# B&R Automation Studio project KeePak_Bliss_Reworked (part 2)

### Types.typ
```iecst
TYPE
	AdhesCtrlInterface_Commands_typ : 	STRUCT
		MelterOn : BOOL;
		MelterStandbyOff : BOOL;
		MelterStandbyOn : BOOL;
		PumpsOn : BOOL;
		PurgeChannel1 : {REDUND_UNREPLICABLE} BOOL;
		PurgeChannel2 : {REDUND_UNREPLICABLE} BOOL;
		PurgeChannel3 : {REDUND_UNREPLICABLE} BOOL;
		PurgeChannel4 : {REDUND_UNREPLICABLE} BOOL;
		WriteChannelTemp : BOOL;
		GlobalTempChanged : BOOL;
	END_STRUCT;
	AdhesCtrlInterface_Pars_typ : 	STRUCT
		SavedPatterns : ARRAY[0..3]OF AdhesivePatternCollections_typ;
		AdhesivePatterns : {REDUND_UNREPLICABLE} ARRAY[0..MAX_NUM_GLUE_CHANNELS_M1]OF AdhesivePattern_typ;
		AdhesiveHMIPatterns : {REDUND_UNREPLICABLE} ARRAY[0..MAX_NUM_GLUE_CHANNELS_M1]OF AdhesivePattern_typ;
		StitchPercentage : {REDUND_UNREPLICABLE} REAL;
		ChannelModulationCtrl : ARRAY[0..MAX_NUM_ONOFF_PATTERNS_M1]OF INT;
		BeadLengths : {REDUND_UNREPLICABLE} ARRAY[0..MAX_NUM_ONOFF_PATTERNS_M1]OF REAL := [4(10)];
		FeedbackIsHardwire : BOOL;
		FeedbackIsModbusTCP : BOOL;
		NordsonComms : NordsonData_typ;
		NordsonFeedbackSelection : NordsonFeedbackSelection_enum;
		NumAdhesiveChannels : {REDUND_UNREPLICABLE} USINT;
		PatternSelection : USINT;
	END_STRUCT;
	AdhesCtrlInterface_Status_typ : 	STRUCT
		AlarmActive : {REDUND_UNREPLICABLE} BOOL;
		ATS_AddOnOverLimit : BOOL;
		ATS_AddOnUnderLimit : BOOL;
		FeederFault : {REDUND_UNREPLICABLE} BOOL;
		GlueApplicationAllowed : {REDUND_UNREPLICABLE} BOOL;
		GlueCyclePos : {REDUND_UNREPLICABLE} REAL;
		LatchedEncoderPos : {REDUND_UNREPLICABLE} REAL;
		LowLevel : {REDUND_UNREPLICABLE} BOOL;
		NordsonInStandby : BOOL;
		ServiceNeeded : {REDUND_UNREPLICABLE} BOOL;
		UnitFault : {REDUND_UNREPLICABLE} BOOL;
		UnitReady : {REDUND_UNREPLICABLE} BOOL;
	END_STRUCT;
	AdhesiveChannelColormaps_typ : 	STRUCT
		Delay : {REDUND_UNREPLICABLE} ARRAY[0..MAX_NUM_ONOFF_PATTERNS_M1]OF USINT;
		Glue : {REDUND_UNREPLICABLE} ARRAY[0..MAX_NUM_ONOFF_PATTERNS_M1]OF USINT;
	END_STRUCT;
	AdhesiveChannelDatapoints_typ : 	STRUCT
		Delay : {REDUND_UNREPLICABLE} ARRAY[0..MAX_NUM_ONOFF_PATTERNS_M1]OF UINT;
		Glue : {REDUND_UNREPLICABLE} ARRAY[0..MAX_NUM_ONOFF_PATTERNS_M1]OF UINT;
		RowLabel : {REDUND_UNREPLICABLE} UINT;
	END_STRUCT;
	AdhesiveCtrlInterface_typ : 	STRUCT
		Commands : {REDUND_UNREPLICABLE} AdhesCtrlInterface_Commands_typ;
		Parameters : {REDUND_UNREPLICABLE} AdhesCtrlInterface_Pars_typ;
		Status : {REDUND_UNREPLICABLE} AdhesCtrlInterface_Status_typ;
	END_STRUCT;
	AdhesivePatternCollections_typ : 	STRUCT
		AdhesivePatterns : ARRAY[0..MAX_NUM_GLUE_CHANNELS_M1]OF AdhesivePattern_typ;
	END_STRUCT;
	AdhesivePattern_typ : 	STRUCT
		DelayDistance : {REDUND_UNREPLICABLE} ARRAY[0..MAX_NUM_ONOFF_PATTERNS_M1]OF REAL;
		GlueOnDistance : {REDUND_UNREPLICABLE} ARRAY[0..MAX_NUM_ONOFF_PATTERNS_M1]OF REAL;
	END_STRUCT;
	AlarmListAdapter_typ : 	STRUCT
		Acknowledged : {REDUND_UNREPLICABLE} ARRAY[0..49]OF STRING[10];
		Active : {REDUND_UNREPLICABLE} ARRAY[0..49]OF STRING[10];
		Code : {REDUND_UNREPLICABLE} ARRAY[0..49]OF STRING[10];
	END_STRUCT;
	AxisInitStates_enum :
		( (*Axis Control States*)
		AXIS_INIT_DONE := 500,
		AXIS_INIT_RETRIEVE_PARS := 10,
		AXIS_INIT_TRANSFER_PARS := 0,
		AXIS_INIT_WAIT_FOR_INIT := 20
		);
	AxisStates_enum :
		( (*Axis Control States*)
		AXIS_STATE_INIT := 0,
		AXIS_STATE_POWERON_PREP := 1,
		AXIS_STATE_POWERON := 2,
		AXIS_STATE_COUPLED := 70,
		AXIS_STATE_ERROR := 999,
		AXIS_STATE_HOME := 30,
		AXIS_STATE_IDLE := 80,
		AXIS_STATE_MOVE := 90,
		AXIS_STATE_MOVE_TO_MASTER := 50,
		AXIS_STATE_MOVE_VELOCITY := 91,
		AXIS_STATE_WAIT_FOR_MASTER_READY := 85,
		AXIS_STATE_W_COUPLE := 60,
		AXIS_STATE_W_HOME := 40,
		AXIS_STATE_POWERSAVER := 100,
		AXIS_STATE_POWERBACK := 101
		);
	Axis_enums :
		( (*Axis enumerations*)
		CCW := 4,
		CC_LEFT := 2,
		CC_RIGHT := 3,
		CSW_LEFT := 0,
		CSW_Left11 := 11,
		CSW_Left12 := 12,
		CSW_Left13 := 13,
		CSW_Left14 := 14,
		CSW_Left15 := 15,
		CSW_Left16 := 16,
		CSW_Left17 := 17,
		CSW_Left18 := 18,
		CSW_Left19 := 19,
		CSW_RIGHT := 1,
		FOLDING_ARM_DA_LEFT := 7,
		FOLDING_ARM_DA_RIGHT := 8,
		FOLDING_BAR := 5,
		FOLDING_TOOL_HA_LEFT := 9,
		FOLDING_TOOL_HA_RIGHT := 10,
		FTCL := 6
		);
	Axis_Interface_Comds_ToMapp_typ : 	STRUCT  (*Axis Commands to Mapp*)
		CoupleToMaster : BOOL;
		Home : BOOL;
		JogNeg : BOOL;
		JogPos : BOOL;
		LoadConfig : BOOL;
		MoveAbs : BOOL;
		MoveAdditive : BOOL;
		MoveVelocity : BOOL;
		Power : BOOL;
		SaveConfig : BOOL;
		Stop : BOOL;
		TorqueLimitingOn : BOOL;
		Update : BOOL;
	END_STRUCT;
	Axis_Interface_Commands_typ : 	STRUCT  (*Axis Commands*)
		Init : BOOL;
		MoveVelocityTrigStop : BOOL;
		RequestCoupleToMaster : BOOL;
		RequestHome : BOOL;
		RequestJogNeg : BOOL;
		RequestJogPos : BOOL;
		RequestMoveAbs : BOOL;
		RequestMoveAdditive : BOOL;
		RequestMoveVelocity : BOOL;
		Stop : USINT;
		ToMapp : Axis_Interface_Comds_ToMapp_typ;
		StartPowerSaver : BOOL;
		StopPowerSaver : BOOL;
	END_STRUCT;
	Axis_Interface_Parameters_typ : 	STRUCT  (*Axis Parameters*)
		AxisAndDrivePars : MpAxisBasicConfigType;
		CouplingMaster : UDINT;
		CouplingParameters : MpAxisCouplingParType;
		MovementParameters : MpAxisBasicParType;
		TriggerDistance : REAL; (*Distance that should be moved after an axis sees a tigger event when using MC_BR_MoveVelocityTriggStop*)
	END_STRUCT;
	Axis_Interface_Status_typ : 	STRUCT  (*Axis Statuses*)
		ActualTorque : LREAL;
		ActualPosition : LREAL;
		ActualSpeed : REAL;
		AxisInitialized : BOOL;
		AxisState : STRING[50];
		ConfigCommandDone : BOOL;
		DefaultRecipeLoaded : BOOL;
		Error : BOOL;
		Homed : BOOL;
		InMotion : BOOL;
		InPosition : BOOL;
		InSync : BOOL;
		MappCommandBusy : BOOL;
		MoveComplete : BOOL;
		PoweredOn : BOOL;
		ReadyToPowerOn : BOOL;
		TriggerMoveDone : BOOL;
		AxisBasicActive : BOOL;
		ClearOfRoller : BOOL;
		PositiveStatusID : USINT; (*The absolute value of the Info.Diag.StatusID.ID from the AxisBasic FUB*)
		StatusSeverity : UDINT;
		StatusCode : UINT;
		InternalID : DINT;
		InternalSeverity : UDINT;
		PositiveInternalFacility : UDINT; (*The absolute value of  Info.Diag.Internal.Facility from the AxisBasic FUB*)
		InternalCode : UINT;
		ExecutingCmd : UDINT;
		PowerSaverModeOn : BOOL;
	END_STRUCT;
	Axis_Interface_typ : 	STRUCT  (*servo Axis Interface*)
		Commands : Axis_Interface_Commands_typ;
		Parameters : Axis_Interface_Parameters_typ;
		Status : Axis_Interface_Status_typ;
	END_STRUCT;
	BitmapSelectDatapoints_typ : 	STRUCT
		AlarmActive : {REDUND_UNREPLICABLE} USINT;
		ResetPress : {REDUND_UNREPLICABLE} BOOL;
		RunPress : {REDUND_UNREPLICABLE} BOOL;
		StopPress : {REDUND_UNREPLICABLE} BOOL;
		VacuumPress : {REDUND_UNREPLICABLE} BOOL;
	END_STRUCT;
	Channel_typ : 	STRUCT
		ActualPressure : REAL;
		PressureSetpoint : REAL;
	END_STRUCT;
	ColorMapDatapoints_typ : 	STRUCT
		AdhesiveChannelsColormaps : {REDUND_UNREPLICABLE} ARRAY[0..MAX_NUM_GLUE_CHANNELS_M1]OF AdhesiveChannelColormaps_typ;
		AdhesiveSystemOK : {REDUND_UNREPLICABLE} USINT;
		AdhesiveUnitFault : {REDUND_UNREPLICABLE} USINT;
		AdhesiveUnitFeederFault : {REDUND_UNREPLICABLE} USINT;
		AdhesiveUnitLevelLow : {REDUND_UNREPLICABLE} USINT;
		AdhesiveUnitReady : {REDUND_UNREPLICABLE} USINT;
		AdhesiveUnitServiceNeeded : {REDUND_UNREPLICABLE} USINT;
		AdhesiveUseageLow : {REDUND_UNREPLICABLE} USINT;
		AirPressureOK : {REDUND_UNREPLICABLE} USINT;
		ATSAddOnOver : USINT;
		ATSAddOnUnder : USINT;
		AutoModeSelected : {REDUND_UNREPLICABLE} USINT;
		DownstreamSensorOK : {REDUND_UNREPLICABLE} USINT;
		DriveFaultOK : {REDUND_UNREPLICABLE} USINT;
		GlueSystemOK : {REDUND_UNREPLICABLE} USINT;
		JogModeSelected : {REDUND_UNREPLICABLE} USINT;
		NordsonEditTemps : USINT;
		RecipeLoaded : {REDUND_UNREPLICABLE} USINT;
		RecipeSystemBusy : {REDUND_UNREPLICABLE} USINT;
		SafetyOK : {REDUND_UNREPLICABLE} USINT;
		VacuumOK : {REDUND_UNREPLICABLE} USINT;
		VacuumPressureOK : {REDUND_UNREPLICABLE} USINT;
		VacuumPumpOn : {REDUND_UNREPLICABLE} USINT;
		Valve1OK : {REDUND_UNREPLICABLE} USINT;
		Valve2OK : {REDUND_UNREPLICABLE} USINT;
		Valve3OK : {REDUND_UNREPLICABLE} USINT;
		Valve4OK : USINT;
	END_STRUCT;
	DigitalInputs_typ : 	STRUCT
		AdhesiveLevelLow : {REDUND_UNREPLICABLE} BOOL;
		AdhesivePhotoEye : {REDUND_UNREPLICABLE} BOOL;
		AdhesivePhotoEye_2 : {REDUND_UNREPLICABLE} BOOL;
		AdhesiveUnitNotFaulted : {REDUND_UNREPLICABLE} BOOL;
		AdhesiveUnitReady : {REDUND_UNREPLICABLE} BOOL;
		AirPressureOK : {REDUND_UNREPLICABLE} BOOL;
		BodyDetect : BOOL;
		DownstreamSensor : {REDUND_UNREPLICABLE} BOOL;
		DownstreamSensorRaw : {REDUND_UNREPLICABLE} BOOL;
		LeftEndDetect : BOOL;
		LowAdhesiveUseage : {REDUND_UNREPLICABLE} BOOL;
		Pneumatics580StatusWord3 : {REDUND_UNREPLICABLE} UINT;
		PnuematicsHWStatusV0 : BOOL;
		PnuematicsHWStatusV2 : BOOL;
		PnuematicsHWStatusV4 : BOOL;
		PnuematicsHWStatusV6 : BOOL;
		RightEndDetect : BOOL;
		SafetyOK : {REDUND_UNREPLICABLE} BOOL;
		SSI_Parallel : {REDUND_UNREPLICABLE} SSI_Paraller_typ;
		VacHigh : BOOL;
		VacLow : BOOL;
		VacuumPressureOK : {REDUND_UNREPLICABLE} BOOL;
		VacuumTempOK : {REDUND_UNREPLICABLE} BOOL;
		X_PickRetracted : BOOL;
		X_PickExtended : BOOL;
		Y_PickRetract : BOOL;
		X_BlowOff : BOOL;
		BodyHopperLow : BOOL;
		LeftHopperLow : BOOL;
		RightHopperLow : BOOL;
		BodyHopperMotor_RUN : BOOL;
		LeftHopperMotor_RUN : BOOL;
		RightHopperMotor_RUN : BOOL;
		LubricationCounter : BOOL;
		BodyHopperMotor_OFF : BOOL;
		LeftHopperMotor_OFF : BOOL;
		RightHopperMotor_OFF : BOOL;
		DownstreamSensorON : BOOL;
		BodyPickHome : BOOL;
		BodyVacuumAchieved : BOOL;
		SidePickVacuumAchieved : BOOL;
		SideFoldSensor : BOOL;
		SideFoldVacuumAchieved : BOOL;
	END_STRUCT;
	DigitalOutputs_typ : 	STRUCT
		AirOn : {REDUND_UNREPLICABLE} BOOL;
		AmberLightStack : {REDUND_UNREPLICABLE} BOOL;
		BlowOffOn : BOOL;
		BottomFolder : {REDUND_UNREPLICABLE} BOOL;
		CompressionAirOn : BOOL;
		GlueChannel1 : {REDUND_UNREPLICABLE} BOOL;
		GlueChannel2 : {REDUND_UNREPLICABLE} BOOL;
		GlueChannel3 : {REDUND_UNREPLICABLE} BOOL;
		GlueChannel4 : {REDUND_UNREPLICABLE} BOOL;
		GreenLightStack : {REDUND_UNREPLICABLE} BOOL;
		HighCompression : BOOL;
		LowCompression : BOOL;
		PickAndPlace_X : BOOL;
		Pneumatics580ControlWord1 : {REDUND_UNREPLICABLE} UINT;
		PnuematicsValve0 : BOOL;
		PnuematicsValve2 : BOOL;
		PnuematicsValve4 : BOOL;
		PnuematicsValve6 : BOOL;
		PushOn : {REDUND_UNREPLICABLE} BOOL;
		RedLightStack : {REDUND_UNREPLICABLE} BOOL;
		ResetEuchner : BOOL;
		ResetSafety : {REDUND_UNREPLICABLE} BOOL;
		TopFolder : {REDUND_UNREPLICABLE} BOOL;
		VacuumOn : {REDUND_UNREPLICABLE} BOOL;
		ZeroEncoder : {REDUND_UNREPLICABLE} BOOL;
		SidePanelVacOn : BOOL;
		SidePanelVacBlowOff : BOOL;
		X_PickSolenoid : BOOL;
		Y_PickSolenoid : BOOL;
		OutConveyorOn_1 : BOOL;
		OutConveyorOn_2 : BOOL;
		OutConveyorOn_3 : BOOL;
		BodyVacuumOn : BOOL;
		BodyKicker : BOOL;
		SidePickCylinder : BOOL;
		LeftSideFoldCylinder : BOOL;
		RightSideFoldCylinder : BOOL;
		SidePanelHoldVacuum : BOOL;
		FoldingHoldVacuum : BOOL;
		CompressionCylinder : BOOL;
	END_STRUCT;
	Encoders_typ : {REDUND_UNREPLICABLE} 	STRUCT
		SickSSIPos : {REDUND_UNREPLICABLE} UDINT;
		SickSSIPosDegrees : {REDUND_UNREPLICABLE} REAL;
		FeedEncoderPos : {REDUND_UNREPLICABLE} UDINT;
		FeedEncoderPosDegrees : {REDUND_UNREPLICABLE} REAL;
		RamEncoderPos : {REDUND_UNREPLICABLE} UDINT;
		RamEncoderPosDegrees : {REDUND_UNREPLICABLE} REAL;
	END_STRUCT;
	FolderTypeSelection_enum :
		(
		FOLDER_LINMOT := 1,
		FOLDER_PNEUMATIC := 0
		);
	FoldpushCtrlInterface_Pars_typ : 	STRUCT
		BottomFolderOffPos : REAL;
		BottomFolderOnPos : REAL;
		FolderTypeSelection : FolderTypeSelection_enum;
		HighCompressionOffPos : REAL;
		HighCompressionOnPos : REAL;
		LinMotBotFolder : LinAxis_typ;
		LinMotTopFolder : LinAxis_typ;
		LowCompressionOffPos : REAL;
		LowCompressionOnPos : REAL;
		NumaticsTypeSelection : NumaticsTypeSelection_enum;
		PushOff : {REDUND_UNREPLICABLE} REAL;
		PushOn : {REDUND_UNREPLICABLE} REAL;
		TopFolderOffPos : REAL;
		TopFolderOnPos : REAL;
	END_STRUCT;
	FoldpushCtrlInterface_Status_typ : 	STRUCT
		BottomFoldValveStatus : {REDUND_UNREPLICABLE} BOOL;
		CompOnValveStatus : BOOL;
		CompressionAllowed : BOOL;
		FoldersActuationAllowed : {REDUND_UNREPLICABLE} BOOL;
		HardwireConfig : BOOL;
		LinMotConfig : BOOL;
		PneumaticConfig : BOOL;
		PowelinkConfig : BOOL;
		PushValveStatus : {REDUND_UNREPLICABLE} BOOL;
		TopFoldValveStatus : {REDUND_UNREPLICABLE} BOOL;
	END_STRUCT;
	FoldPushCtrlInterface_typ : 	STRUCT
		Commands : {REDUND_UNREPLICABLE} FoldPushCtrlInt_Commands_typ;
		Parameters : {REDUND_UNREPLICABLE} FoldpushCtrlInterface_Pars_typ;
		Status : {REDUND_UNREPLICABLE} FoldpushCtrlInterface_Status_typ;
	END_STRUCT;
	FoldPushCtrlInt_Commands_typ : 	STRUCT
		placehold : {REDUND_UNREPLICABLE} BOOL;
	END_STRUCT;
	HMIControl_Commands_typ : 	STRUCT
		CancelBoxChange : BOOL;
		ConfirmBoxChange : BOOL;
		CycleBodyHopper : BOOL;
		CycleLeftHopper : BOOL;
		CycleRightHopper : BOOL;
		CycleServoRam : BOOL;
		CycleServoPnP : BOOL;
		HomeServoFeed : BOOL;
		HomeBodyHopper : BOOL;
		HomeLeftHopper : BOOL;
		HomeRightHopper : BOOL;
		HomeServoRam : BOOL;
		HomeServoPnP : BOOL;
		JogForward : BOOL;
		JogReverse : BOOL;
		JogServoFeedNeg : BOOL;
		JogServoFeedPos : BOOL;
		JogBodyHopperNeg : BOOL;
		JogBodyHopperPos : BOOL;
		JogLeftHopperNeg : BOOL;
		JogLeftHopperPos : BOOL;
		JogRightHopperNeg : BOOL;
		JogRightHopperPos : BOOL;
		JogServoRamNeg : BOOL;
		JogServoRamPos : BOOL;
		JogServoPnPNeg : BOOL;
		JogServoPnPPos : BOOL;
		LoadRecipe : BOOL;
		LoadRecipeType1 : BOOL;
		LoadRecipeType2 : BOOL;
		RequestBoxType1 : BOOL;
		RequestBoxType2 : BOOL;
		RequestReset : BOOL;
		RequestStop : BOOL;
		RequestVacuumOn : BOOL;
		RequestVFDRun : BOOL;
		SaveRecipe : BOOL;
		SelectAutoMode : BOOL;
		SelectJogMode : BOOL;
		StartServoFeed : BOOL;
		StartBodyHopper : BOOL;
		StartLeftHopper : BOOL;
		StartRightHopper : BOOL;
		ZeroEncoder : BOOL;
		EnableShowMode : BOOL;
	END_STRUCT;
	HMIControl_Parameters_typ : 	STRUCT
		ServoFeedAccel : REAL;
		ServoFeedJogVelocity : REAL;
		ServoFeedTorqueLimit : REAL;
		ServoFeedVelocity : REAL;
		BodyHopperAccel : REAL;
		BodyHopperEndDwellTime : UDINT;
		BodyHopperEndPosition : REAL;
		BodyHopperJogVelocity : REAL;
		BodyHopperStartDwellTime : UDINT;
		BodyHopperStartPosition : REAL;
		BodyHopperTorqueLimit : REAL;
		BodyHopperVelocity : REAL;
		BodyKickerTime : UDINT;
		BodyKickerRetractTime : UDINT;
		LeftHopperAccel : REAL;
		LeftHopperEndDwellTime : UDINT;
		LeftHopperEndPosition : REAL;
		LeftHopperJogVelocity : REAL;
		LeftHopperStartDwellTime : UDINT;
		LeftHopperStartPosition : REAL;
		LeftHopperTorqueLimit : REAL;
		LeftHopperVelocity : REAL;
		RightHopperAccel : REAL;
		RightHopperEndDwellTime : UDINT;
		RightHopperEndPosition : REAL;
		RightHopperJogVelocity : REAL;
		RightHopperStartDwellTime : UDINT;
		RightHopperStartPosition : REAL;
		RightHopperTorqueLimit : REAL;
		RightHopperVelocity : REAL;
		ServoRamAccel : REAL;
		ServoRamEndDwellTime : UDINT;
		ServoRamSidePickTime : UDINT;
		ServoRamSidePickRetractTime : UDINT;
		ServoRamSideFoldTime : UDINT;
		ServoRamSideFoldRetractTime : UDINT;
		ServoRamEndPosition : REAL;
		ServoRamFoldStartPos : REAL;
		ServoRamFoldEndPos : REAL;
		ServoRamJogVelocity : REAL;
		ServoRamStartDwellTime : UDINT;
		ServoRamStartPosition : REAL;
		ServoRamTorqueLimit : REAL;
		ServoRamNegativeVelocity : REAL;
		ServoRamSideFormingVelocity : REAL;
		ServoRamBoxFormingVelocity : REAL;
		ServoRamClearPosition : REAL;
		ServoRamMiddlePosition : REAL;
		ServoPnPAccel : REAL;
		ServoPnPEndDwellTime : UDINT;
		ServoPnPEndPosition : REAL;
		ServoPnPVacuumOffPosition : REAL;
		ServoPnPJogVelocity : REAL;
		ServoPnPStartDwellTime : UDINT;
		ServoPnPStartPosition : REAL;
		ServoPnPTorqueLimit : REAL;
		ServoPnPNegativeVelocity : REAL;
		ServoPnPPositiveVelocity : REAL;
		PickAndPlaceDwell : UDINT;
		BodyHopperDwellTime : UDINT;
		LeftHopperDwellTime : UDINT;
		RightHopperDwellTime : UDINT;
		BodyHopperTimeoutTime : UDINT;
		LeftHopperTimeoutTime : UDINT;
		RightHopperTimeoutTime : UDINT;
		ServoRamTimeoutTime : UDINT;
		ServoRamPowerSaverTime : UDINT;
		AtTorqueTime : UDINT;
		PickDwellTime : UDINT;
		TopFeedJamTime : UDINT;
		VacuumOffTime : UDINT;
		DownPulseTime : UDINT;
		Y_DelayTime : UDINT;
		BlowOffTime : UDINT;
		SetCycleCount : UDINT;
		LubeCycleCount : UDINT;
		LowFeedJamTime : UDINT;
		LowHopperTime : UDINT;
		LowBodyHopperTime : UDINT;
		LowLeftHopperTime : UDINT;
		LowRightHopperTime : UDINT;
		RamDelay : UDINT;
	END_STRUCT;
	HMIControl_typ : 	STRUCT
		BitmapSelectDatapoints : {REDUND_UNREPLICABLE} BitmapSelectDatapoints_typ;
		ColorMapDatapoints : {REDUND_UNREPLICABLE} ColorMapDatapoints_typ;
		Commands : {REDUND_UNREPLICABLE} HMIControl_Commands_typ;
		Parameters : HMIControl_Parameters_typ;
		StatusDatapoints : {REDUND_UNREPLICABLE} StatusDatapoints_typ;
	END_STRUCT;
	Home_Parameters_typ : 	STRUCT  (*Axis Homing Parameters*)
		ServoFeed : MpAxisHomingType;
		BodyHopper : MpAxisHomingType;
		LeftHopper : MpAxisHomingType;
		RightHopper : MpAxisHomingType;
		ServoRam : MpAxisHomingType;
		ServoPnP : MpAxisHomingType;
	END_STRUCT;
	IO_typ : 	STRUCT
		DIs : {REDUND_UNREPLICABLE} DigitalInputs_typ;
		DOs : {REDUND_UNREPLICABLE} DigitalOutputs_typ;
		Encoders : {REDUND_UNREPLICABLE} Encoders_typ;
		ModuleOKs : {REDUND_UNREPLICABLE} ARRAY[0..99]OF BOOL;
		SafetyStatus : SafetyStatus_typ;
	END_STRUCT;
	LightStack_typ :
		(
		LIGHTSTACK_PATLITE := 1,
		LIGHTSTACK_TRI := 0
		);
	LinAxisCommand_typ : 	STRUCT  (*Axis command type*)
		ErrorReset : BOOL; (*Reset error command*)
		Home : BOOL; (*Home command*)
		HomeRequest : BOOL; (*Request for home from HMI*)
		JogNegative : BOOL; (*Jog neg command*)
		JogNegativeRequest : BOOL; (*Request for jog negative*)
		JogPositive : BOOL; (*Jog pos command*)
		JogPositiveRequest : BOOL; (*Request for jog positive*)
		MoveAbsolute : BOOL; (*Move absolute command*)
		MoveAbsoluteRequest : BOOL; (*Request for move absolute*)
		MoveAdditive : BOOL; (*Move additive command*)
		Power : BOOL; (*Power command*)
		SaveConfig : BOOL;
		Stop : BOOL; (*Stop command*)
	END_STRUCT;
	LinAxisParameter_typ : 	STRUCT  (*Axis parameter type*)
		ExtendAccel : REAL;
		ExtendDecel : REAL;
		ExtendPos : LREAL;
		ExtendSpeed : REAL;
		MpBasicConfig : MpAxisBasicConfigType; (*Axis configuration parameters for change at runtime*)
		MpBasicParameters : MpAxisBasicParType; (*Mp params*)
		RetractAccel : REAL;
		RetractDecel : REAL;
		RetractPos : LREAL;
		RetractSpeed : REAL;
	END_STRUCT;
	LinAxisStatus_typ : 	STRUCT  (*Axis status type*)
		EndlessPosValid : BOOL; (*Endless position is valid*)
		Error : BOOL; (*Error active on axis*)
		ErrorId : DINT; (*Error id*)
		HomeCheck : BOOL;
		Info : MpAxisBasicInfoType;
		InPosition : BOOL; (*Axis in position*)
		IsHomed : BOOL; (*Axis is homed*)
		MoveActive : BOOL; (*Move is active on the axis*)
		Position : LREAL; (*Current position of axis*)
		PowerOn : BOOL; (*Axis is on*)
		Ready : BOOL; (*Axis is in standstill and homed*)
		Stopped : BOOL; (*Axis is stopped*)
		Velocity : REAL; (*Current velocity of axis*)
	END_STRUCT;
	LinAxis_typ : 	STRUCT  (*Axis type*)
		Command : LinAxisCommand_typ; (*Command*)
		Parameter : LinAxisParameter_typ; (*Parameter*)
		Status : LinAxisStatus_typ; (*Status*)
	END_STRUCT;
	LinMotState_enum :
		(
		STATE_ERROR,
		STATE_HOME_CHECK,
		STATE_HOME_RESTORE,
		STATE_HOME_STANDBY,
		STATE_HOME_TORQUE,
		STATE_INIT,
		STATE_IS_HOMED,
		STATE_JOG_NEG,
		STATE_JOG_POS,
		STATE_MOVE,
		STATE_READY
		);
	ModeCtrlInterface_Commands_typ : {REDUND_UNREPLICABLE} 	STRUCT
		ForceSafetyReset : {REDUND_UNREPLICABLE} BOOL;
		Reset : {REDUND_UNREPLICABLE} BOOL;
		Run : {REDUND_UNREPLICABLE} BOOL;
		SetAutoMode : {REDUND_UNREPLICABLE} BOOL;
		SetJogMode : {REDUND_UNREPLICABLE} BOOL;
		Stop : {REDUND_UNREPLICABLE} BOOL;
		SetShowMode : {REDUND_UNREPLICABLE} BOOL;
	END_STRUCT;
	ModeCtrlInterface_Parameters_typ : 	STRUCT
		BottomSensor : BOOL;
		DownstreamClear : UDINT := 1000;
		DownstreamIgnored : BOOL;
		DownstreamTimeout : UDINT := 1000;
		DwellTime : {REDUND_UNREPLICABLE} UDINT;
		InPositionTolerance : REAL := 10.0;
		LightStackSelection : LightStack_typ;
		MachineType : USINT;
		MaxPPM : UINT;
		MinPPM : UINT;
		PiecesPerMinute : {REDUND_UNREPLICABLE} UINT;
		SideSensors : BOOL;
		StopPosition : {REDUND_UNREPLICABLE} REAL;
		VaccumStopTime : UDINT := 200;
		SidePickTime : UDINT;
	END_STRUCT;
	ModeCtrlInterface_Status_typ : 	STRUCT
		AtStopPosition : {REDUND_UNREPLICABLE} BOOL;
		BlissPanelAlarmActive : BOOL;
		Dwelling : {REDUND_UNREPLICABLE} BOOL;
		DwellModeEnabled : {REDUND_UNREPLICABLE} BOOL;
		InAutoMode : {REDUND_UNREPLICABLE} BOOL;
		InBlissPanelWindow : BOOL;
		Jogging : {REDUND_UNREPLICABLE} BOOL;
		MachineIsBliss : BOOL;
		Running : {REDUND_UNREPLICABLE} BOOL;
		WaitingOnDownstream : BOOL;
	END_STRUCT;
	ModeCtrlInterface_typ : 	STRUCT
		Commands : {REDUND_UNREPLICABLE} ModeCtrlInterface_Commands_typ;
		Parameters : {REDUND_UNREPLICABLE} ModeCtrlInterface_Parameters_typ;
		Status : ModeCtrlInterface_Status_typ;
	END_STRUCT;
	NordsonData_typ : 	STRUCT
		AdhesiveUsePerHour : UDINT;
		Alert : BOOL;
		ByPassFeedback : BOOL;
		ChannelActTemp : ARRAY[0..NUM_NORDSON_TEMP_ZONES_M1]OF UINT;
		ChannelDataCmpResult : DINT;
		ChannelDataSize : UDINT;
		ChannelSetTempActual : ARRAY[0..NUM_NORDSON_TEMP_ZONES_M1]OF UINT;
		ChannelSetTempRequested : ARRAY[0..NUM_NORDSON_TEMP_ZONES_M1]OF UINT;
		CommFault : BOOL;
		CommFaultInDataValue : BOOL;
		ConsecutiveErrorCount : USINT;
		FeedbackTime : TIME := T#1s;
		HeatUpPhaseActive : BOOL;
		HoseSetTemp : UINT;
		MelterIsOn : BOOL;
		MelterStatus : UINT;
		PumpStartUpProtectionOn : BOOL;
		ShutDown : BOOL;
		StandbyTimeoutTime : TIME := T#2h;
		TempUnit : USINT;
		UnitFaulted : BOOL;
		UnitReady : BOOL;
		GlobalSetTemp : UINT;
	END_STRUCT;
	NordsonFeedbackSelection_enum :
		(
		NORDSON_HARDWIRE := 0,
		NORDSON_MODBUSTCP := 1
		);
	NordsonRxPacket_typ : 	STRUCT
		Byte0_1_Status : UINT;
		Byte2_Ack_Data_Index : USINT;
		Byte3_Ack_Channel_Num : USINT;
		Byte4_5_Read_Data_0 : UINT;
		Byte6_7_Read_Data_1 : UINT;
		Byte8_9_Read_Data_2 : UINT;
		Byte10_11_Read_Data_3 : UINT;
		Byte12_13_Read_Data_4 : UINT;
		Byte14_15_Read_Data_5 : UINT;
	END_STRUCT;
	NordsonTxPacket_typ : 	STRUCT
		Byte0_MelterControl : USINT;
		Byte1_Command : USINT;
		Byte2_Data_Index : USINT;
		Byte3_Channel_Num : USINT;
		Byte4_5_WriteData : UINT;
		Byte6_7_Mot1Spd : UINT;
		Byte8_9_Mot2Spd : UINT;
		Byte10_11_Mot3Spd : UINT;
		Byte12_13_Mot4Spd : UINT;
		Byte14_15_NotUsed : UINT;
	END_STRUCT;
	NumaticsTypeSelection_enum :
		(
		NUMATICS_HARDWIRE,
		NUMATICS_POWERLINK
		);
	RamControlInterface_typ : 	STRUCT
		Commands : {REDUND_UNREPLICABLE} RamCtrlInterface_Commands_typ;
		Parameters : {REDUND_UNREPLICABLE} RamCtrlInterface_Parameters_typ;
		Status : {REDUND_UNREPLICABLE} RamCtrlInterface_Status_typ;
	END_STRUCT;
	RamCtrlInterface_Commands_typ : 	STRUCT
		Home : {REDUND_UNREPLICABLE} BOOL;
		JogNegative : {REDUND_UNREPLICABLE} BOOL;
		JogPositive : {REDUND_UNREPLICABLE} BOOL;
		MoveAbsolute : {REDUND_UNREPLICABLE} BOOL;
		MoveAdditive : {REDUND_UNREPLICABLE} BOOL;
		MoveVelocity : {REDUND_UNREPLICABLE} BOOL;
		PowerOn : {REDUND_UNREPLICABLE} BOOL;
		VFDAlarmReset : {REDUND_UNREPLICABLE} BOOL;
	END_STRUCT;
	RamCtrlInterface_Parameters_typ : 	STRUCT
		Acceleration : {REDUND_UNREPLICABLE} REAL;
		CurrentLimit : {REDUND_UNREPLICABLE} REAL;
		GearRatio : REAL := 54;
		JogSpeed : {REDUND_UNREPLICABLE} REAL;
		Position : {REDUND_UNREPLICABLE} REAL;
	END_STRUCT;
	RamCtrlInterface_Status_typ : 	STRUCT
		ActualPosition : {REDUND_UNREPLICABLE} LREAL;
		ActualSpeed : {REDUND_UNREPLICABLE} LREAL;
		AlarmActive : {REDUND_UNREPLICABLE} BOOL;
		DriveSpeed : {REDUND_UNREPLICABLE} INT;
		Home : {REDUND_UNREPLICABLE} BOOL;
		InPosition : {REDUND_UNREPLICABLE} BOOL;
		MotorCurrent : {REDUND_UNREPLICABLE} UINT;
		MoveActive : {REDUND_UNREPLICABLE} BOOL;
		Position : {REDUND_UNREPLICABLE} REAL;
		PoweredOn : {REDUND_UNREPLICABLE} BOOL;
		Running : {REDUND_UNREPLICABLE} BOOL;
		Stopped : BOOL;
		STOStatus : UINT;
		VFDAlarmDetected : {REDUND_UNREPLICABLE} BOOL;
		VFDAlarmNumber : {REDUND_UNREPLICABLE} INT;
		VFDAlarmText : {REDUND_UNREPLICABLE} STRING[80];
	END_STRUCT;
	RecipeCtrlInterface_Commands_typ : 	STRUCT
		ChangeRecipe : BOOL;
		LoadRecipe : {REDUND_UNREPLICABLE} BOOL;
		SaveRecipe : {REDUND_UNREPLICABLE} BOOL;
	END_STRUCT;
	RecipeCtrlInterface_Pars_typ : 	STRUCT
		RecipeIndex : USINT;
		RecipeName : {REDUND_UNREPLICABLE} STRING[100];
	END_STRUCT;
	RecipeCtrlInterface_Status_typ : 	STRUCT
		Busy : {REDUND_UNREPLICABLE} BOOL;
		LoadedRecipeIndex : USINT;
		LoadedRecipeName : {REDUND_UNREPLICABLE} STRING[255];
		RecipeHasBeenLoaded : BOOL;
	END_STRUCT;
	RecipeCtrlInterface_typ : 	STRUCT
		Commands : {REDUND_UNREPLICABLE} RecipeCtrlInterface_Commands_typ;
		Parameters : {REDUND_UNREPLICABLE} RecipeCtrlInterface_Pars_typ;
		Status : {REDUND_UNREPLICABLE} RecipeCtrlInterface_Status_typ;
	END_STRUCT;
	Register_typ : 	STRUCT
		ChannelActualPressureWord : UDINT;
		ChannelSetPressureWord : UDINT;
		TankActualLevelWord : UINT;
	END_STRUCT;
	SafetyStatus_typ : 	STRUCT
		BackEstopOK : BOOL;
		CabinetEStopStatus : UINT;
		FrontEStopOK : BOOL;
		GuardDoorsOK : BOOL;
		SafetyProgramRunning : BOOL;
	END_STRUCT;
	SSI_Paraller_typ : {REDUND_UNREPLICABLE} 	STRUCT
		Bits : {REDUND_UNREPLICABLE} ARRAY[0..15]OF BOOL;
		FeedBits : {REDUND_UNREPLICABLE} ARRAY[0..15]OF BOOL;
		RamBits : {REDUND_UNREPLICABLE} ARRAY[0..15]OF BOOL;
	END_STRUCT;
	StatusDatapoints_typ : 	STRUCT
		AdhesiveChannelSDPs : {REDUND_UNREPLICABLE} ARRAY[0..MAX_NUM_GLUE_CHANNELS_M1]OF AdhesiveChannelDatapoints_typ;
		AdhesivePatternDialogSDP : UINT := 1;
		AdhesivePatternConfirmDialogSDP : UINT := 1;
		AdhesivePatternConfirmedSDP : UINT;
		AdhesiveUnitFaultSDP : {REDUND_UNREPLICABLE} UINT;
		AdhesiveUnitLevelLowSDP : {REDUND_UNREPLICABLE} UINT;
		AdhesiveUnitNotReadySDP : {REDUND_UNREPLICABLE} UINT;
		AdhesiveUseageLowSDP : {REDUND_UNREPLICABLE} UINT;
		AutoModeSDP : {REDUND_UNREPLICABLE} UINT;
		BlissSDP : UINT;
		HardwireValveSDP : USINT;
		JogStatusDatapoint : {REDUND_UNREPLICABLE} UINT;
		LinMotBotHomeSDP : UINT;
		LinMotSDP : UINT;
		LinMotTopHomeSDP : UINT;
		LinMotTuningSDP : UINT;
		MaintenanceSDP : {REDUND_UNREPLICABLE} UINT;
		MotorVacuumSDP : UINT;
		NordsonModbusSDP : UINT;
		NordsonStandbyOffSDP : UINT;
		PnuematicFolderSDP : UINT;
		RecipeDialogSDP : UINT;
		RecipeIndexSDP : UINT;
		RecipeReq1SDP : UINT;
		RecipeReq2SDP : UINT;
		RestartInhibitSDP : UINT;
		SafetyStartingSDP : UINT;
		ServoLayerSDP : {REDUND_UNREPLICABLE} UINT;
		ServoRamHomeSDP : UINT;
		SmartVacuumLayerSDP : {REDUND_UNREPLICABLE} UINT;
		TraySDP : UINT;
		VacuumPressureFaultSDP : {REDUND_UNREPLICABLE} UINT;
		VenturiVacuumSDP : UINT;
		ZeroEncoderSDP : {REDUND_UNREPLICABLE} UINT;
		HopperLowSDP : UINT;
		HomeServoRamSDP : UINT;
		LubeSDP : UINT;
		BodyHopperSwitchSDP : UINT;
		LeftHopperSwitchSDP : UINT;
		RightHopperSwitchSDP : UINT;
	END_STRUCT;
	Tank_typ : 	STRUCT
		ActualLevel : REAL;
	END_STRUCT;
	VacCtrlConfig_enum :
		(
		VAC_MOTOR := 0,
		VAC_VENTURI := 1
		);
	VacCtrlInterface_Commands_typ : 	STRUCT
		BlowOffOnManual : BOOL;
		VacuumOn : {REDUND_UNREPLICABLE} BOOL;
		VenturiOn : BOOL;
		VenturiOnManual : BOOL;
	END_STRUCT;
	VacCtrlInterface_Parameters_typ : 	STRUCT
		BlowOffTime : UINT;
		ManualVenturiVacuumOff : BOOL;
		VacConfig : VacCtrlConfig_enum;
		VacOffPos : REAL;
		VacOnPos : REAL;
	END_STRUCT;
	VacCtrlInterface_Status_typ : 	STRUCT
		AlarmActive : {REDUND_UNREPLICABLE} BOOL;
		Pressure : {REDUND_UNREPLICABLE} REAL;
		StandstillTimout : BOOL;
		StandstillTimoutSet : BOOL;
		VacLowAlarm : BOOL;
		VacLowCycle : BOOL;
	END_STRUCT;
	VacCtrlInterface_typ : 	STRUCT
		Commands : {REDUND_UNREPLICABLE} VacCtrlInterface_Commands_typ;
		Parameters : {REDUND_UNREPLICABLE} VacCtrlInterface_Parameters_typ;
		Status : {REDUND_UNREPLICABLE} VacCtrlInterface_Status_typ;
	END_STRUCT;
END_TYPE
```

### Program Logical/ModeControl/ModeControl_ST

#### Types.typ
```iecst
TYPE
	BlissSideCheckStates_enum :
		(
		SIDE_CHECK_IDLE,
		SIDE_CHECK_FIRST_CYCLE,
		SIDE_CHECK_LOOK_FOR_EYE,
		SIDE_CHECK_EYE_FOUND,
		SIDE_CHECK_EYE_MISSED
		);
	BlissBodyCheckStates_enum :
		(
		BODY_CHECK_IDLE,
		BODY_CHECK_FIRST_CYCLE,
		BODY_CHECK_LOOK_FOR_EYE,
		BODY_CHECK_EYE_FOUND,
		BODY_CHECK_EYE_MISSED
		);
END_TYPE
```

#### Variables.var
```iecst
VAR
	AirPressureAlarmActive : BOOL;
	AirPressureNotOK : BOOL;
	AirPressureNotOKTimer : TON;
	BlowOff_Pulse : TP;
	BlowOff_Trigger : BOOL;
	BodyCheckError : BOOL;
	BodyCheckErrorActive : BOOL;
	BodyHopperLowAlarm : BOOL;
	BodyHopperLowTMR : TON;
	BodyPanelTimeout : TON;
	BoxPickTMR : TON;
	CountReset : BOOL;
	DistanceFromStopPosition : REAL;
	DownstreamBlocked : BOOL;
	DownstreamSensorONTimer : TON;
	DownstreamSensorTimer : TON;
	Dummy : BOOL;
	DwellTimer : TON;
	EuchnerSafeResetTimer : TON;
	FeedPosFinal : LREAL;
	FeedPositionCapture : LREAL;
	FeedServoPosSP : LREAL;
	FeedServoTimeout : BOOL;
	FeedServoTMR : TON;
	FeedStopTimer : TON;
	ForceBodyPanellError : BOOL;
	FrontEStopNotOKActive : BOOL;
END_VAR
VAR CONSTANT
	Ftrig_BlowOffOnManual : F_TRIG := (0); (*Falling edge detection function block for this variable*)
END_VAR
VAR
	Ftrig_DownstreamBlocked : F_TRIG;
	GluePhotoEyeAlarmActive : BOOL;
	GuardDoorNotOKActive : BOOL;
	HopperRunningError : BOOL;
	InBlissSidePanelCheckWindow : BOOL;
	InfeedCheckError : BOOL;
	InfeedTimeout : TON;
	LeftHopperLowAlarm : BOOL;
	LeftHopperLowTMR : TON;
	LubeReset : BOOL;
	LubricationCounter : CTU;
	MoveVelocityRequest : BOOL;
	OldEncoderPos : REAL;
	PhotoEyeCheckErrorActive : BOOL;
	PhotoEyeTimeout : TON;
	PickAndPlaceDwelling : BOOL;
	PickAndPlaceDwellTimer : TON;
	PickAndPlaceHasBox : BOOL;
	PickDwellTime : TIME;
	PnPTimeout : TON;
	PnPTimeoutError : BOOL;
	RamAtStopPosition : BOOL;
	RamCycleCount : UDINT;
	RearEStopNotOKActive : BOOL;
	Return_Trigger : BOOL;
	RightHopperLowAlarm : BOOL;
	RightHopperLowTMR : TON;
	Rtrig_AlarmActive : R_TRIG; (*Rising edge detection function block for this variable*)
	Rtrig_BlowOffManual : R_TRIG; (*Rising edge detection function block for this variable*)
	Rtrig_BlowOffTrigger : R_TRIG; (*Rising edge detection function block for this variable*)
	Rtrig_DownstreamBlocked : R_TRIG; (*Rising edge detection function block for this variable*)
	Rtrig_FeedServoTMR : R_TRIG; (*Rising edge detection function block for this variable*)
	Rtrig_HopperLow : R_TRIG; (*Rising edge detection function block for this variable*)
	Rtrig_InfeedBoxPresent : R_TRIG; (*Rising edge detection function block for this variable*)
	Rtrig_LubricationCounter : R_TRIG; (*Rising edge detection function block for this variable*)
	Rtrig_PhotoEyeSeen : R_TRIG; (*Rising edge detection function block for this variable*)
	Rtrig_RequestStop : R_TRIG; (*Rising edge detection function block for this variable*)
	Rtrig_RequestVFDRun : R_TRIG;
	SafetyNotOKActive : BOOL;
	SafetyResetRequestTimer : TON;
	ShowModeTimer : TON;
	SideCheckError : BOOL;
	SideCheckErrorActive : BOOL;
	status : UDINT;
	StopFeedServo : BOOL;
	StopPositionDwellExpire : BOOL;
	StopTriggerByDownstream : BOOL;
	TON_BlowOff : TON; (*Timer for blow off after vacuum is shut off (user defined time)*)
	TON_RamDelay : TON; (*Timer for the Ram to delay forward motion*)
	VaccumStopTimer : TON;
	VacuumOffTime : TIME;
	VacuumTimer : TON;
	Vacuum_ON : BOOL;
	Y_Delay : TON;
	Y_Down_Pulse : TP;
	Y_Trigger : BOOL;
END_VAR
```

#### Cyclic1.st
```iecst
PROGRAM _CYCLIC
	(* Insert code here *)

    // HMI Glue pattern inputs are in inches, but the code needs mm
    gAdhesiveCtrlInterface.Parameters.AdhesivePatterns[0].DelayDistance[0] := gAdhesiveCtrlInterface.Parameters.AdhesiveHMIPatterns[0].DelayDistance[0] * 25.4;
    gAdhesiveCtrlInterface.Parameters.AdhesivePatterns[0].DelayDistance[1] := gAdhesiveCtrlInterface.Parameters.AdhesiveHMIPatterns[0].DelayDistance[1] * 25.4;
    gAdhesiveCtrlInterface.Parameters.AdhesivePatterns[0].DelayDistance[2] := gAdhesiveCtrlInterface.Parameters.AdhesiveHMIPatterns[0].DelayDistance[2] * 25.4;
    gAdhesiveCtrlInterface.Parameters.AdhesivePatterns[0].DelayDistance[3] := gAdhesiveCtrlInterface.Parameters.AdhesiveHMIPatterns[0].DelayDistance[3] * 25.4;
    gAdhesiveCtrlInterface.Parameters.AdhesivePatterns[1].DelayDistance[0] := gAdhesiveCtrlInterface.Parameters.AdhesiveHMIPatterns[1].DelayDistance[0] * 25.4;
    gAdhesiveCtrlInterface.Parameters.AdhesivePatterns[1].DelayDistance[1] := gAdhesiveCtrlInterface.Parameters.AdhesiveHMIPatterns[1].DelayDistance[1] * 25.4;
    gAdhesiveCtrlInterface.Parameters.AdhesivePatterns[1].DelayDistance[2] := gAdhesiveCtrlInterface.Parameters.AdhesiveHMIPatterns[1].DelayDistance[2] * 25.4;
    gAdhesiveCtrlInterface.Parameters.AdhesivePatterns[1].DelayDistance[3] := gAdhesiveCtrlInterface.Parameters.AdhesiveHMIPatterns[1].DelayDistance[3] * 25.4;
    gAdhesiveCtrlInterface.Parameters.AdhesivePatterns[2].DelayDistance[0] := gAdhesiveCtrlInterface.Parameters.AdhesiveHMIPatterns[2].DelayDistance[0] * 25.4;
    gAdhesiveCtrlInterface.Parameters.AdhesivePatterns[2].DelayDistance[1] := gAdhesiveCtrlInterface.Parameters.AdhesiveHMIPatterns[2].DelayDistance[1] * 25.4;
    gAdhesiveCtrlInterface.Parameters.AdhesivePatterns[2].DelayDistance[2] := gAdhesiveCtrlInterface.Parameters.AdhesiveHMIPatterns[2].DelayDistance[2] * 25.4;
    gAdhesiveCtrlInterface.Parameters.AdhesivePatterns[2].DelayDistance[3] := gAdhesiveCtrlInterface.Parameters.AdhesiveHMIPatterns[2].DelayDistance[3] * 25.4;
    gAdhesiveCtrlInterface.Parameters.AdhesivePatterns[3].DelayDistance[0] := gAdhesiveCtrlInterface.Parameters.AdhesiveHMIPatterns[3].DelayDistance[0] * 25.4;
    gAdhesiveCtrlInterface.Parameters.AdhesivePatterns[3].DelayDistance[1] := gAdhesiveCtrlInterface.Parameters.AdhesiveHMIPatterns[3].DelayDistance[1] * 25.4;
    gAdhesiveCtrlInterface.Parameters.AdhesivePatterns[3].DelayDistance[2] := gAdhesiveCtrlInterface.Parameters.AdhesiveHMIPatterns[3].DelayDistance[2] * 25.4;
    gAdhesiveCtrlInterface.Parameters.AdhesivePatterns[3].DelayDistance[3] := gAdhesiveCtrlInterface.Parameters.AdhesiveHMIPatterns[3].DelayDistance[3] * 25.4;

    gAdhesiveCtrlInterface.Parameters.AdhesivePatterns[0].GlueOnDistance[0] := gAdhesiveCtrlInterface.Parameters.AdhesiveHMIPatterns[0].GlueOnDistance[0] * 25.4;
    gAdhesiveCtrlInterface.Parameters.AdhesivePatterns[0].GlueOnDistance[1] := gAdhesiveCtrlInterface.Parameters.AdhesiveHMIPatterns[0].GlueOnDistance[1] * 25.4;
    gAdhesiveCtrlInterface.Parameters.AdhesivePatterns[0].GlueOnDistance[2] := gAdhesiveCtrlInterface.Parameters.AdhesiveHMIPatterns[0].GlueOnDistance[2] * 25.4;
    gAdhesiveCtrlInterface.Parameters.AdhesivePatterns[0].GlueOnDistance[3] := gAdhesiveCtrlInterface.Parameters.AdhesiveHMIPatterns[0].GlueOnDistance[3] * 25.4;
    gAdhesiveCtrlInterface.Parameters.AdhesivePatterns[1].GlueOnDistance[0] := gAdhesiveCtrlInterface.Parameters.AdhesiveHMIPatterns[1].GlueOnDistance[0] * 25.4;
    gAdhesiveCtrlInterface.Parameters.AdhesivePatterns[1].GlueOnDistance[1] := gAdhesiveCtrlInterface.Parameters.AdhesiveHMIPatterns[1].GlueOnDistance[1] * 25.4;
    gAdhesiveCtrlInterface.Parameters.AdhesivePatterns[1].GlueOnDistance[2] := gAdhesiveCtrlInterface.Parameters.AdhesiveHMIPatterns[1].GlueOnDistance[2] * 25.4;
    gAdhesiveCtrlInterface.Parameters.AdhesivePatterns[1].GlueOnDistance[3] := gAdhesiveCtrlInterface.Parameters.AdhesiveHMIPatterns[1].GlueOnDistance[3] * 25.4;
    gAdhesiveCtrlInterface.Parameters.AdhesivePatterns[2].GlueOnDistance[0] := gAdhesiveCtrlInterface.Parameters.AdhesiveHMIPatterns[2].GlueOnDistance[0] * 25.4;
    gAdhesiveCtrlInterface.Parameters.AdhesivePatterns[2].GlueOnDistance[1] := gAdhesiveCtrlInterface.Parameters.AdhesiveHMIPatterns[2].GlueOnDistance[1] * 25.4;
    gAdhesiveCtrlInterface.Parameters.AdhesivePatterns[2].GlueOnDistance[2] := gAdhesiveCtrlInterface.Parameters.AdhesiveHMIPatterns[2].GlueOnDistance[2] * 25.4;
    gAdhesiveCtrlInterface.Parameters.AdhesivePatterns[2].GlueOnDistance[3] := gAdhesiveCtrlInterface.Parameters.AdhesiveHMIPatterns[2].GlueOnDistance[3] * 25.4;
    gAdhesiveCtrlInterface.Parameters.AdhesivePatterns[3].GlueOnDistance[0] := gAdhesiveCtrlInterface.Parameters.AdhesiveHMIPatterns[3].GlueOnDistance[0] * 25.4;
    gAdhesiveCtrlInterface.Parameters.AdhesivePatterns[3].GlueOnDistance[1] := gAdhesiveCtrlInterface.Parameters.AdhesiveHMIPatterns[3].GlueOnDistance[1] * 25.4;
    gAdhesiveCtrlInterface.Parameters.AdhesivePatterns[3].GlueOnDistance[2] := gAdhesiveCtrlInterface.Parameters.AdhesiveHMIPatterns[3].GlueOnDistance[2] * 25.4;
    gAdhesiveCtrlInterface.Parameters.AdhesivePatterns[3].GlueOnDistance[3] := gAdhesiveCtrlInterface.Parameters.AdhesiveHMIPatterns[3].GlueOnDistance[3] * 25.4;

    //SAFETY CHECKS 0001
    IF NOT gAlarmSystemActive THEN
        RETURN;
    END_IF

    //AIR PRESSURE ON/NOK 0002
    //Do not set air pressure alarm unless air pressure has been low for 20 seconds
    AirPressureNotOKTimer.PT := T#20s;
    AirPressureNotOKTimer.IN := (NOT gIO.DIs.AirPressureOK AND NOT gIsSimulated);
    AirPressureNotOKTimer();
    AirPressureNotOK         := AirPressureNotOKTimer.Q;

    //MP ALARMX CHECK STATE AIR PRESSURE LOW 0003
    AirPressureAlarmActive := MpAlarmXCheckState(gAlarmXCore, ALARM_AIR_PRESSURE_LOW, mpALARMX_STATE_ACTIVE);

    //MP ALARMX SET/RESET AIR PRESSURE LOW 0004 AND 0005
    //Set/clear air pressure alarm
    IF (AirPressureNotOK AND NOT AirPressureAlarmActive) THEN
        status := MpAlarmXSet(gAlarmXCore,ALARM_AIR_PRESSURE_LOW);
    ELSIF (NOT AirPressureNotOK AND AirPressureAlarmActive) THEN
        status := MpAlarmXReset(gAlarmXCore,ALARM_AIR_PRESSURE_LOW);
    END_IF

    //MP ALARMX CHECK STATE SAFETY OK/NOK 0006
    SafetyNotOKActive := MpAlarmXCheckState(gAlarmXCore, ALARM_SAFETY_NOTOK, mpALARMX_STATE_ACTIVE);

    //MP ALARMX SET/RESET SAFETY OK/NOK 0007 AND 0008
    //Set/Clear Safety Alarm
    IF (NOT gIO.DIs.SafetyOK AND NOT SafetyNotOKActive AND gIO.SafetyStatus.SafetyProgramRunning) THEN
        status := MpAlarmXSet(gAlarmXCore,ALARM_SAFETY_NOTOK);
    ELSIF (gIO.DIs.SafetyOK AND SafetyNotOKActive AND gIO.SafetyStatus.SafetyProgramRunning) THEN
        status := MpAlarmXReset(gAlarmXCore,ALARM_SAFETY_NOTOK);
    END_IF

    //MP ALARMX CHECK STATE GUARD DOOR 0009
    GuardDoorNotOKActive := MpAlarmXCheckState(gAlarmXCore, ALARM_SAFETY_GUARD_DOOR, mpALARMX_STATE_ACTIVE);

    //MP ALARMX SET/RESET GUARD DOORS 0010 AND 0011
    //Set/Clear Safety Alarm
    IF (NOT gIO.SafetyStatus.GuardDoorsOK AND NOT GuardDoorNotOKActive AND gIO.SafetyStatus.SafetyProgramRunning) THEN
        status := MpAlarmXSet(gAlarmXCore,ALARM_SAFETY_GUARD_DOOR);
    ELSIF (gIO.SafetyStatus.GuardDoorsOK AND GuardDoorNotOKActive AND gIO.SafetyStatus.SafetyProgramRunning) THEN
        status := MpAlarmXReset(gAlarmXCore,ALARM_SAFETY_GUARD_DOOR);
    END_IF

    //MP ALARMX CHECK STATE FRONT ESTOP 0012
    FrontEStopNotOKActive := MpAlarmXCheckState(gAlarmXCore, ALARM_SAFETY_FRONT_ESTOP, mpALARMX_STATE_ACTIVE);

    //MP ALARMX SET/RESET FRONT ESTOP 0013 AND 0014
    //Set/Clear Safety Alarm
    IF (NOT gIO.SafetyStatus.FrontEStopOK AND NOT FrontEStopNotOKActive AND gIO.SafetyStatus.SafetyProgramRunning) THEN
        status := MpAlarmXSet(gAlarmXCore,ALARM_SAFETY_FRONT_ESTOP);
    ELSIF (gIO.SafetyStatus.FrontEStopOK AND FrontEStopNotOKActive AND gIO.SafetyStatus.SafetyProgramRunning) THEN
        status := MpAlarmXReset(gAlarmXCore,ALARM_SAFETY_FRONT_ESTOP);
    END_IF

    //MP ALARMX CHECK STATE REAR ESTOP 0015
    RearEStopNotOKActive := MpAlarmXCheckState(gAlarmXCore, ALARM_SAFETY_REAR_ESTOP, mpALARMX_STATE_ACTIVE);

    //MP ALARMX SET/RESET REAR ESTOP 0016 AND 0017
    //Set/Clear Safety Alarm
    IF (NOT gIO.SafetyStatus.BackEstopOK AND NOT RearEStopNotOKActive AND gIO.SafetyStatus.SafetyProgramRunning) THEN
        status := MpAlarmXSet(gAlarmXCore,ALARM_SAFETY_REAR_ESTOP);
    ELSIF (gIO.SafetyStatus.BackEstopOK AND RearEStopNotOKActive AND gIO.SafetyStatus.SafetyProgramRunning) THEN
        status := MpAlarmXReset(gAlarmXCore,ALARM_SAFETY_REAR_ESTOP);
    END_IF

    //TURN AIR ON 0018
    //If safety is OK, Turn air On and turn off the red light
    gIO.DOs.AirOn         := gIO.DIs.SafetyOK;
    gIO.DOs.RedLightStack := NOT (gIO.DIs.SafetyOK AND NOT gModeControlInterface.Status.BlissPanelAlarmActive);

    //NO ALARMS GREEN LIGHT 0019
    //If there are no alarms active, turn on the green light
    gIO.DOs.GreenLightStack := NOT gAlarmActive;

    //ALARM YELLOW LIGHT 0020
    //If there is an active alarm, or the hopper is low, turn on yellow stack light
    gIO.DOs.AmberLightStack := (gAlarmActive OR gIO.DIs.BodyHopperLow);

	//DO NOT FINISH CYCLE OF ANYTHING OTHER THAN STOP BUTTON IS PRESSED 0024
	//If an alarm is active or safety is not ok or jog mode is selected, do not finish the selected cycle
	IF (gServoFeedInterface.Status.Error OR gBodyHopperInterface.Status.Error OR gLeftHopperInterface.Status.Error OR gRightHopperInterface.Status.Error OR gServoRamInterface.Status.Error OR
		NOT gIO.DIs.SafetyOK OR gHMI.Commands.SelectJogMode OR gHighSeverityAlarmActive OR BodyCheckError) THEN
		PickAndPlaceHasBox                         := FALSE;
		PickAndPlaceDwelling                       := FALSE;
		PhotoEyeSeen                               := FALSE;
		Vacuum_ON                                  := FALSE;
		gIO.DOs.X_PickSolenoid                     := FALSE;
		gIO.DOs.BlowOffOn                          := FALSE;
	END_IF

	//DOES NOT LET MACHINE RUN IF GLUE SYSTEM HAS AN ERROR 0025
	//Do not allow machine to run if glue system has an alarm (Removed gLowSeverityAlarmActive)
	IF (gAdhesiveCtrlInterface.Status.AlarmActive OR
		gServoFeedInterface.Status.Error OR gBodyHopperInterface.Status.Error OR gLeftHopperInterface.Status.Error OR gRightHopperInterface.Status.Error OR gServoRamInterface.Status.Error OR
		gLowSeverityAlarmActive OR gHighSeverityAlarmActive OR gServoPnPInterface.Status.Error) THEN
		gHMI.Commands.RequestVFDRun := FALSE;
	END_IF

	//AUTO MODE RUN REQUEST FINISH CYCLE 0026
	//If we're in auto mode, and run request has been made or we should finish the running, set move request
	MoveVelocityRequest := (gHMI.Commands.SelectAutoMode AND gHMI.Commands.RequestVFDRun);

	//RAM POSITION AND STOP POSITION (360-0 ROLLOVER)DetermineDistanceToStopPos 0027
	DistanceFromStopPosition := DetermineDistanceToStopPos(gIO.Encoders.FeedEncoderPos, gModeControlInterface.Parameters.StopPosition);

	//KEEPS SERVOS RUNNING TO FINISH CYCLE 0030
	//VFD run command was the run command for the old machine. Keep servos cycling while it is true
	gHMI.Commands.StartBodyHopper := gHMI.Commands.RequestVFDRun;
	gHMI.Commands.StartLeftHopper := gHMI.Commands.RequestVFDRun;
	gHMI.Commands.StartRightHopper := gHMI.Commands.RequestVFDRun;
	gHMI.Commands.StartServoFeed   := (gHMI.Commands.RequestVFDRun (*AND NOT DownstreamBlocked*) AND NOT StopFeedServo);
	gHMI.Commands.CycleServoRam    := gHMI.Commands.RequestVFDRun;
	gHMI.Commands.CycleServoPnP    := gHMI.Commands.RequestVFDRun;
	// The discharge conveyor is controlled by three bits.
	// If #1 is on, then it is running slow. If #1 and #3 are on, then it is running medium speed. #2 Can be used if we need a faster speed.
	gIO.DOs.OutConveyorOn_1 := gHMI.Commands.RequestVFDRun OR (gCyclesToFinish > 0);
	gIO.DOs.OutConveyorOn_2 := gHMI.Commands.RequestVFDRun OR (gCyclesToFinish > 0);
	gIO.DOs.OutConveyorOn_3 := gHMI.Commands.RequestVFDRun OR (gCyclesToFinish > 0);

	//RISING EDGE FOR SERVOINPUT SIGNAL 0031
	Rtrig_FeedServoTMR(CLK := FeedServoTMR.Q);
	StopFeed := Rtrig_FeedServoTMR.Q;

	//0032 SERVO RAM TRIGGER SET IN FEED HANDLER. COMMENTED OUT

	//HOPPER LOW ALARMS 0033
	BodyHopperLowTMR.IN := gIO.DIs.BodyHopperLow;
    BodyHopperLowTMR.PT := gHMI.Parameters.LowBodyHopperTime;
    BodyHopperLowTMR();
    IF BodyHopperLowTMR.Q THEN
        BodyHopperLowAlarm := TRUE;
	END_IF
	LeftHopperLowTMR.IN := gIO.DIs.LeftHopperLow;
	LeftHopperLowTMR.PT := gHMI.Parameters.LowLeftHopperTime;
	LeftHopperLowTMR();
	IF LeftHopperLowTMR.Q THEN
		LeftHopperLowAlarm := TRUE;
	END_IF
	RightHopperLowTMR.IN := gIO.DIs.RightHopperLow;
	RightHopperLowTMR.PT := gHMI.Parameters.LowRightHopperTime;
	RightHopperLowTMR();
	IF RightHopperLowTMR.Q THEN
		RightHopperLowAlarm := TRUE;
	END_IF

    //FEED STOP TIMER 0034
    //Timer for the HopperLows to trigger StopFeed
    FeedStopTimer.IN := gIO.DIs.BodyHopperLow OR gIO.DIs.RightHopperLow OR gIO.DIs.LeftHopperLow;
    FeedStopTimer.PT := gHMI.Parameters.LowHopperTime;
    FeedStopTimer();
    HoperLowStop     := FeedStopTimer.Q;

    //HOPPER LOW ALARM RESET 0035
    IF NOT gIO.DIs.BodyHopperLow THEN
        BodyHopperLowAlarm := FALSE;
	END_IF
	IF NOT gIO.DIs.LeftHopperLow THEN
		LeftHopperLowAlarm := FALSE;
	END_IF
	IF NOT gIO.DIs.RightHopperLow THEN
		RightHopperLowAlarm := FALSE;
	END_IF

	//==========================================================================================================================================================

	//Downstream Sensor Timer Addition 02/11/2025
	//DownstreamSensorTimer.PT := gModeControlInterface.Parameters.DownstreamTimeout;
	//DownstreamSensorTimer.IN := (gIO.DIs.DownstreamSensorRaw AND NOT gModeControlInterface.Parameters.DownstreamIgnored);
	//DownstreamSensorTimer();
	//IF DownstreamSensorTimer.Q THEN
	//	gIO.DIs.DownstreamSensor := TRUE;
	//END_IF

	//DownstreamBlocked := gIO.DIs.DownstreamSensor AND RamAtStopPosition;
	//gModeControlInterface.Status.WaitingOnDownstream := MoveVelocityRequest AND DownstreamBlocked;

	// Downsream Sensor Timer Addition 02/11/2025
	DownstreamSensorTimer.PT := gModeControlInterface.Parameters.DownstreamTimeout;
	DownstreamSensorTimer.IN := (gIO.DIs.DownstreamSensorRaw AND NOT gModeControlInterface.Parameters.DownstreamIgnored);
	DownstreamSensorTimer();
	gIO.DIs.DownstreamSensor := DownstreamSensorTimer.Q;
	DownstreamBlocked := gIO.DIs.DownstreamSensor AND gRamAtStopPosition;
	IF MoveVelocityRequest AND DownstreamBlocked THEN
		gModeControlInterface.Status.WaitingOnDownstream := TRUE;
		gHMI.Commands.RequestVFDRun := FALSE;
	END_IF
	// If waiting on downstream but the downstream has cleared, then start running
	IF gModeControlInterface.Status.WaitingOnDownstream AND NOT gIO.DIs.DownstreamSensor THEN
		gModeControlInterface.Status.WaitingOnDownstream := FALSE;
		gHMI.Commands.RequestVFDRun := TRUE;
		// Otherwise, if the stop button is pressed, clear the waiting signal
	ELSIF gHMI.Commands.RequestStop THEN
		gModeControlInterface.Status.WaitingOnDownstream := FALSE;
	END_IF

	//==========================================================================================================================================================

	//PHOTO EYES SETTING AND RESETTING
	IF (gIO.DIs.AdhesivePhotoEye) THEN
		PhotoEyeSeen := TRUE;
	END_IF
    IF gIO.DIs.BodyDetect THEN
        PhotoEyeSeen := FALSE;
    END_IF

    //0047
    //Latch the encoder position. this marks the start of the glue cycle
    Rtrig_PhotoEyeSeen(CLK := PhotoEyeSeen);
    IF (Rtrig_PhotoEyeSeen.Q AND ((gHMI.Commands.SelectAutoMode AND gHMI.Commands.RequestVFDRun) OR (gCyclesToFinish > 0))) THEN
        gAdhesiveCtrlInterface.Status.LatchedEncoderPos := LREAL_TO_REAL(gServoFeedInterface.Status.ActualPosition);
        DistanceAfterLatch                              := 0;
        OldEncoderPos                                   := LREAL_TO_REAL(gServoFeedInterface.Status.ActualPosition);
    END_IF

    //0048
    //Determine how far the ram has moved since the photo eye was last seen
    DistanceAfterLatch := (ComputeDistanceMoved(LREAL_TO_REAL(gServoFeedInterface.Status.ActualPosition),OldEncoderPos) + DistanceAfterLatch);

    //0049
    OldEncoderPos := LREAL_TO_REAL(gServoFeedInterface.Status.ActualPosition);

	//BODY PANEL TIMEOUT 0052
	//If the machine is running and a box has passed the photoeyes, but hasn't cleared the photo eye for LowFeedJamTime amount of time, then raise an alarm
    BodyPanelTimeout.PT := gHMI.Parameters.LowFeedJamTime;
    BodyPanelTimeout.IN := (gHMI.Commands.RequestVFDRun AND gIO.DIs.BodyDetect);
    BodyPanelTimeout();
    IF BodyPanelTimeout.Q THEN
        BodyCheckError := TRUE;
    ELSIF gHMI.Commands.RequestReset THEN
        BodyCheckError := FALSE;
	END_IF

	//INFEED TIMEOUT
	//If the machine is running and a box hasnt passed the photoeyes for LowFeedJamTime amount of time, then raise an alarm
	InfeedTimeout.PT := gHMI.Parameters.TopFeedJamTime;
	InfeedTimeout.IN := (gHMI.Commands.RequestVFDRun AND NOT gIO.DIs.BodyDetect);
	InfeedTimeout();
	IF InfeedTimeout.Q THEN
		InfeedCheckError := TRUE;
	ELSIF gHMI.Commands.RequestReset THEN
		InfeedCheckError := FALSE;
	END_IF

    //0053 AND 0054 LUBE COUNTER
    LubricationOK := (LubeCount < gHMI.Parameters.SetCycleCount);

    Rtrig_LubricationCounter(CLK := gIO.DIs.LubricationCounter);
    LubricationCounter.CU    := Rtrig_LubricationCounter.Q;
    LubricationCounter.RESET := LubeReset;
    LubricationCounter.PV    := UDINT_TO_UINT(gHMI.Parameters.LubeCycleCount);
    LubricationCounter();
    CountReset               := LubricationCounter.Q;

    //0055 COUNT AND LUBE COUNT RESET
    LubeReset := CountReset;
    IF CountReset THEN
        LubeCount := 0;
	END_IF

	//make it a fault if the system is reuqested to run while any hopper is off
	IF gHMI.Commands.RequestVFDRun AND (gIO.DIs.LeftHopperMotor_OFF OR gIO.DIs.RightHopperMotor_OFF OR gIO.DIs.BodyHopperMotor_OFF) THEN
		HopperRunningError := TRUE;
	ELSIF gHMI.Commands.RequestReset THEN
		HopperRunningError := FALSE;
	END_IF

    //Disabled this due to the error triggering and not clearing after a few hours
//    PnPTimeout.PT := T#3600s;
//    PnPTimeout.IN := NOT gHMI.Commands.RequestVFDRun AND (gHMI.Commands.RequestStop OR gServoPnPInterface.Status.PoweredOn);
//    PnPTimeout();
 //   IF PnPTimeout.Q THEN
//        PnPTimeoutError := TRUE;
//    ELSIF gHMI.Commands.RequestReset THEN
//        PnPTimeoutError := FALSE;
//    END_IF

	END_PROGRAM
```

#### Init.st
```iecst
PROGRAM _INIT

	gPassword;
	gUserLevel;
	gIO;

	//set these DI's true. physical IO will take over once program runs,
	//and we need to make sure we see a falling edge on these IO points so that alarms are reported
	gIO.DIs.SafetyOK := TRUE;
	gIO.SafetyStatus.BackEstopOK := TRUE;
	gIO.SafetyStatus.FrontEStopOK := TRUE;
	gIO.SafetyStatus.GuardDoorsOK := TRUE;
	gIO.DIs.AirPressureOK := TRUE;
	gIO.DIs.VacuumPressureOK := TRUE;
	gIO.DIs.AdhesiveUnitNotFaulted := TRUE;
	gIO.DIs.AdhesiveUnitReady := TRUE;
	gIO.DIs.AdhesiveLevelLow := FALSE;
	gIO.DIs.VacuumTempOK := TRUE;
	gIO.DIs.BodyHopperLow := TRUE;
	gIO.DIs.LeftHopperLow := TRUE;
	gIO.DIs.RightHopperLow := TRUE;

	gAutoTune := FALSE;
	gCurrentLimitHit := FALSE;

	//PickDwellTime := T#
	gHMI.Parameters.PickDwellTime :=0; //Only Used With Older Style Machines
	gHMI.Parameters.PickAndPlaceDwell := 750; //750ms How Long It Takes To Grab A Box
	gHMI.Parameters.LowHopperTime := 2000; //2S Hopper Low Timer
	gHMI.Parameters.LowFeedJamTime := 10000; // 3S Bottom Photo Eye
	gHMI.Parameters.TopFeedJamTime := 10000; // 10S Top Photo Eyes
	gHMI.Parameters.VacuumOffTime := 1000; // 1S Vacuum Off Time
	gHMI.Parameters.DownPulseTime := 1000; // 1S Only Used On Y Axis Machines
	gHMI.Parameters.Y_DelayTime := 500; // 500ms Only Used On Y Axis Machines
	gHMI.Parameters.BlowOffTime := 100; // 100ms Blow Off and Vacuum Off Trigger
	gHMI.Parameters.LubeCycleCount := 5; // 5 cycles Lube Counter
	gHMI.Parameters.SetCycleCount := 25000; // 25000 Ram Servo Cycles

END_PROGRAM
```

### Program Logical/Recipes/Recipes

#### Cyclic.ld
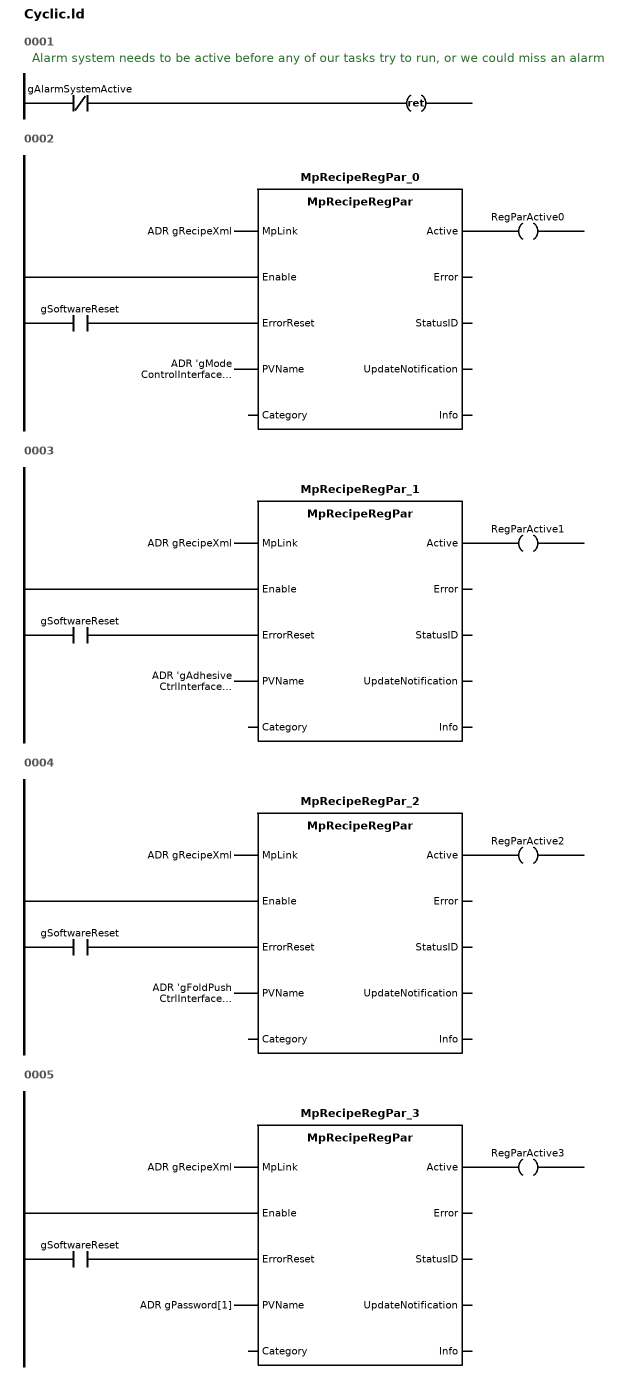
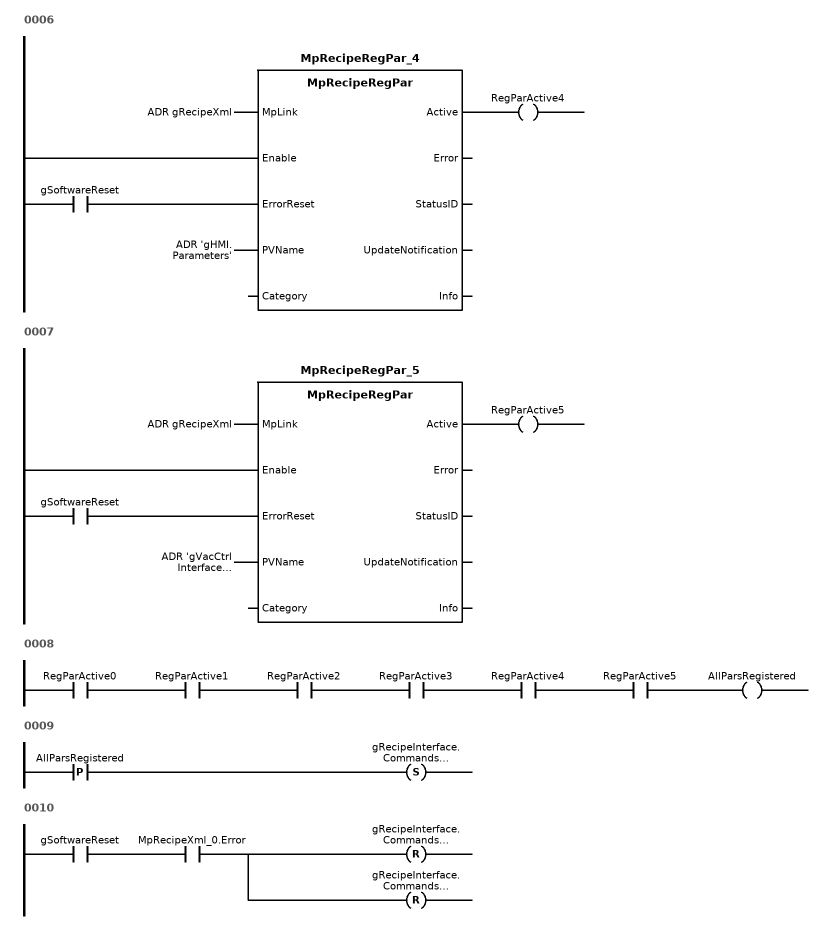
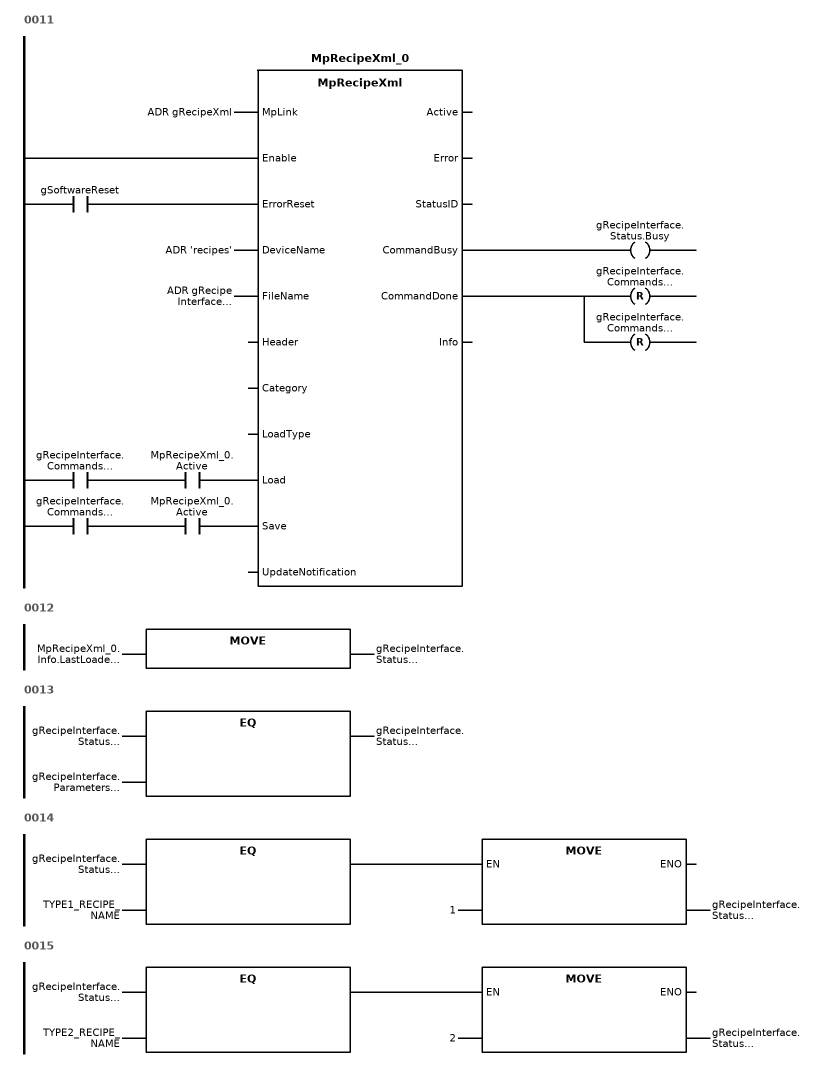
Ladder, written as Structured Text:
```iecst
PROGRAM _CYCLIC
VAR
    _e1 : R_TRIG;
    _p2 : BOOL;
    _p3 : BOOL;
END_VAR
(* Network 1: Alarm system needs to be active before any of our tasks try to run, or we could miss an alarm *)
IF NOT gAlarmSystemActive THEN RETURN; END_IF;

(* Network 2 *)
MpRecipeRegPar_0(MpLink := ADR(gRecipeXml), Enable := TRUE, ErrorReset := gSoftwareReset, PVName := ADR('gModeControlInterface.Parameters'));
RegParActive0 := MpRecipeRegPar_0.Active;

(* Network 3 *)
MpRecipeRegPar_1(MpLink := ADR(gRecipeXml), Enable := TRUE, ErrorReset := gSoftwareReset, PVName := ADR('gAdhesiveCtrlInterface.Parameters'));
RegParActive1 := MpRecipeRegPar_1.Active;

(* Network 4 *)
MpRecipeRegPar_2(MpLink := ADR(gRecipeXml), Enable := TRUE, ErrorReset := gSoftwareReset, PVName := ADR('gFoldPushCtrlInterface.Parameters'));
RegParActive2 := MpRecipeRegPar_2.Active;

(* Network 5 *)
MpRecipeRegPar_3(MpLink := ADR(gRecipeXml), Enable := TRUE, ErrorReset := gSoftwareReset, PVName := ADR(gPassword[1]));
RegParActive3 := MpRecipeRegPar_3.Active;

(* Network 6 *)
MpRecipeRegPar_4(MpLink := ADR(gRecipeXml), Enable := TRUE, ErrorReset := gSoftwareReset, PVName := ADR('gHMI.Parameters'));
RegParActive4 := MpRecipeRegPar_4.Active;

(* Network 7 *)
MpRecipeRegPar_5(MpLink := ADR(gRecipeXml), Enable := TRUE, ErrorReset := gSoftwareReset, PVName := ADR('gVacCtrlInterface.Parameters'));
RegParActive5 := MpRecipeRegPar_5.Active;

(* Network 8 *)
AllParsRegistered := RegParActive0 AND RegParActive1 AND RegParActive2 AND RegParActive3 AND RegParActive4 AND RegParActive5;

(* Network 9 *)
_e1(CLK := AllParsRegistered);
IF _e1.Q THEN gRecipeInterface.Commands.LoadRecipe := TRUE; END_IF;

(* Network 10 *)
IF gSoftwareReset AND MpRecipeXml_0.Error THEN
    gRecipeInterface.Commands.LoadRecipe := FALSE;
    gRecipeInterface.Commands.SaveRecipe := FALSE;
END_IF;

(* Network 11 *)
MpRecipeXml_0(MpLink := ADR(gRecipeXml), Enable := TRUE, ErrorReset := gSoftwareReset, DeviceName := ADR('recipes'), FileName := ADR(gRecipeInterface.Parameters.RecipeName), Load := gRecipeInterface.Commands.LoadRecipe AND MpRecipeXml_0.Active, Save := gRecipeInterface.Commands.SaveRecipe AND MpRecipeXml_0.Active);
gRecipeInterface.Status.Busy := MpRecipeXml_0.CommandBusy;
IF MpRecipeXml_0.CommandDone THEN
    gRecipeInterface.Commands.LoadRecipe := FALSE;
    gRecipeInterface.Commands.SaveRecipe := FALSE;
END_IF;

(* Network 12 *)
gRecipeInterface.Status.LoadedRecipeName := MpRecipeXml_0.Info.LastLoadedRecipe;

(* Network 13 *)
gRecipeInterface.Status.RecipeHasBeenLoaded := gRecipeInterface.Status.LoadedRecipeName = gRecipeInterface.Parameters.RecipeName;

(* Network 14 *)
_p2 := gRecipeInterface.Status.LoadedRecipeName = TYPE1_RECIPE_NAME;
IF _p2 THEN gRecipeInterface.Status.LoadedRecipeIndex := 1; END_IF;

(* Network 15 *)
_p3 := gRecipeInterface.Status.LoadedRecipeName = TYPE2_RECIPE_NAME;
IF _p3 THEN gRecipeInterface.Status.LoadedRecipeIndex := 2; END_IF;
END_PROGRAM
```

### ServoMotionPackGlobal.var
```iecst
VAR
	BodyGrabFailAlarm : BOOL;
	SideGrabFailAlarm : BOOL;
	SideFoldFailAlarm : BOOL;
END_VAR
```

### Program Logical/ServoMotion/ServoRamHandler (IEC)

#### Main.st
```iecst
PROGRAM _INIT

	// Velocities and Accels
	gHMI.Parameters.ServoRamJogVelocity := 50;

	gHMI.Parameters.ServoRamSideFormingVelocity := 500.0;
	gHMI.Parameters.ServoRamBoxFormingVelocity := 750.0;
	gHMI.Parameters.ServoRamNegativeVelocity := 750.0;

	gHMI.Parameters.ServoRamAccel := 2000.0; //values much higher than this create an audible pop sound as tension changes direction in the belt at end of travel

	// Positions
	gHMI.Parameters.ServoRamStartPosition := 14.72;
	gHMI.Parameters.ServoRamMiddlePosition := 255.0;
	gHMI.Parameters.ServoRamFoldStartPos := 75.0;
	gHMI.Parameters.ServoRamFoldEndPos := 290.0;
	gHMI.Parameters.ServoRamEndPosition := 1200.0;

	// Times
	gHMI.Parameters.ServoRamEndDwellTime := 100;
	gHMI.Parameters.ServoRamStartDwellTime := 100;
	gHMI.Parameters.ServoRamSidePickTime:= 300;
	gHMI.Parameters.ServoRamSidePickRetractTime := 300;
	gHMI.Parameters.ServoRamSideFoldTime:= 100;
	gHMI.Parameters.ServoRamSideFoldRetractTime := 50;
	gHMI.Parameters.RamDelay := 100;
	gHMI.Parameters.ServoRamTimeoutTime := 120000;

	// Other
	gHMI.Parameters.ServoRamTorqueLimit := 6.0;
	gHMI.Parameters.ServoRamClearPosition := 300;

	//	gHMI.Parameters.ServoRamTimeoutTime := T#3s;

	gPassword; //need to use this somewhere. Was getting thrown out in slimmed down test code for servo ram

END_PROGRAM

PROGRAM _CYCLIC

	IF gHighSeverityAlarmActive THEN
		state := SERVORAM_ERROR;
	END_IF

	gIO.DOs.ResetSafety := gHMI.Commands.RequestReset OR ForceSafetyReset;

	// Resetting clears the grab and fold alarms
	IF gHMI.Commands.RequestReset THEN
		SideGrabFailAlarm := FALSE;
		SideFoldFailAlarm := FALSE;
		ResetTimeoutAlarm := FALSE;
	END_IF

	// Automatically disable all timers. Explicitly set them in state machine when needed
	EndDwellTimer.IN := FALSE;
	SidePickTimer.IN := FALSE;
	SidePickRetractTimer.IN := FALSE;
	SideFoldTimer.IN := FALSE;
	SideFoldRetractTimer.IN := FALSE;
	RamDelayTimer.IN := FALSE;
	ResetTimeoutTimer.IN := FALSE;

//	// If the hopper has been reset but the machine isn't running, only let the hopper run for an alotted time to protect the motor
//	IF NOT gHMI.Commands.CycleServoRam AND NOT gServoRamInterface.Status.Error AND gServoRamInterface.Status.PoweredOn THEN
//		ResetTimeoutTimer.IN := TRUE;
//	END_IF
//	IF ResetTimeoutTimer.Q THEN
//			ResetTimeoutAlarm := TRUE;
//	END_IF
//	// Resetting clears the timeout alarms
//	IF gHMI.Commands.RequestReset THEN
//		ResetTimeoutAlarm := FALSE;
//		ResetTimeoutTimer.IN := FALSE;
//	END_IF

	IF gServoRamInterface.Status.ActualPosition <= gHMI.Parameters.ServoRamClearPosition THEN
		gServoRamInterface.Status.ClearOfRoller := TRUE;
	ELSE
		gServoRamInterface.Status.ClearOfRoller := FALSE;
	END_IF

//	IF NOT gHMI.Commands.CycleServoRam AND NOT ExerciseRam AND state <> SERVORAM_ERROR AND gServoRamInterface.Status.Homed THEN
//		state := SERVORAM_IDLE;
//	END_IF

	CASE state OF

		SERVORAM_WAIT_FOR_HOME:

			// Servo ram should home automatically on machine start up.
			IF gServoRamInterface.Status.Homed AND ServoRamFirstHomeExecuted THEN
				ServoRamAutoHome := FALSE;
				gRamAtStopPosition := TRUE;
				gHMI.Commands.CycleServoRam := FALSE;
				gServoRamInterface.Commands.ToMapp.TorqueLimitingOn := TRUE; //turn torque limiting on
				state := SERVORAM_IDLE;
			ELSIF gServoRamInterface.Status.PoweredOn AND NOT ServoRamFirstHomeExecuted THEN
				ServoRamAutoHome := TRUE;
				state := SERVORAM_WAIT_FOR_AUTO_HOME;
			END_IF

		SERVORAM_WAIT_FOR_AUTO_HOME:

			IF gServoRamInterface.Status.Homed AND ServoRamFirstHomeExecuted THEN
				ServoRamAutoHome := FALSE;
				gRamAtStopPosition := TRUE;
				gHMI.Commands.CycleServoRam := FALSE;
				gServoRamInterface.Commands.ToMapp.TorqueLimitingOn := TRUE; //turn torque limiting on
				state := SERVORAM_IDLE;
			END_IF

		SERVORAM_IDLE:

			ServoRamAutoHome := FALSE;
			gServoRamInterface.Status.MoveComplete := FALSE; //if we force a transition to IDLE while moving, we may have a stuck move complete flag. clear it here

			gCyclesToFinish := 0;

			// Wait for the ram to be homed and for run to be pressed, then move to the starting position
			IF gHMI.Commands.CycleServoRam AND ServoRamFirstHomeExecuted THEN
				ServoRamBusy := TRUE;
				gRamWaitingOnBox := TRUE; //tell the PnP that we are waiting on a box
				gServoRamInterface.Commands.ToMapp.TorqueLimitingOn := TRUE; //turn torque limiting on
				gServoRamInterface.Parameters.MovementParameters.Position := gHMI.Parameters.ServoRamStartPosition;
				gServoRamInterface.Parameters.MovementParameters.Velocity := gHMI.Parameters.ServoRamNegativeVelocity;
				gServoRamInterface.Commands.RequestMoveAbs := TRUE;
				gRamAtStopPosition := FALSE;
				ServoRamBusy := TRUE;
				state := SERVORAM_MOVE_TO_START;

				//allow the ram to cycle through the start, middle, and end positions. Lets us exercise the movements without using actuators
				//this should only be used to test the machine
			ELSIF ExerciseRam THEN
				gServoRamInterface.Commands.ToMapp.TorqueLimitingOn := TRUE; //turn torque limiting on
				gServoRamInterface.Parameters.MovementParameters.Position := gHMI.Parameters.ServoRamStartPosition;
				gServoRamInterface.Parameters.MovementParameters.Velocity := gHMI.Parameters.ServoRamNegativeVelocity;
				gServoRamInterface.Commands.RequestMoveAbs := TRUE;
				state := SERVORAM_MOVE_TO_START_EX;
			END_IF

		SERVORAM_MOVE_TO_START:

			// At the starting position, turn on the side vacuum and push the cylinders out to grab the side panels
			// The left and right hoppers must be on, the feed wheels must be running, and the PNP must have left its home position
			IF NOT gHMI.Commands.CycleServoRam AND gServoRamInterface.Status.MoveComplete AND (gCyclesToFinish = 0) THEN
				gServoRamInterface.Status.MoveComplete := FALSE;
				gRamAtStopPosition := TRUE;
				state := SERVORAM_IDLE;
			ELSIF gServoRamInterface.Status.MoveComplete AND gIO.DIs.LeftHopperMotor_RUN AND gIO.DIs.RightHopperMotor_RUN AND gIO.DIs.BodyHopperMotor_RUN AND
				gServoFeedInterface.Status.InMotion AND NOT gIO.DIs.BodyPickHome (*AND gIO.DIs.BodyVacuumAchieved*) AND (gCyclesToFinish > 0) THEN
				gRamAtStopPosition := TRUE;
				gServoRamInterface.Status.MoveComplete := FALSE;
				ServoRamBusy := FALSE;
				gIO.DOs.SidePanelVacOn := TRUE;
				gIO.DOs.SidePanelHoldVacuum := TRUE;
				gIO.DOs.SidePickCylinder := TRUE;
				state := SERVORAM_PICK_SIDES;
			END_IF

		SERVORAM_PICK_SIDES:
			SidePickTimer.IN := TRUE;
			// Wait for the side pick timer, then retract the side pick
			IF SidePickTimer.Q THEN
				gIO.DOs.SidePickCylinder := FALSE;
				SidePickRetractTimer.IN := TRUE;
			END_IF
			// When the side pick is retracted, check for side panels
			IF SidePickRetractTimer.Q THEN
				SidePickTimer.IN := FALSE;
				SidePickRetractTimer.IN := FALSE;
				state := SERVORAM_CHECK_FOR_SIDES;
			END_IF

		SERVORAM_CHECK_FOR_SIDES:
			IF gIO.DIs.SidePickVacuumAchieved THEN
				// If the side pick has vacuum, then the sides were picked, move to middle position
				SideFailureCount := 0;
				state := SERVORAM_WAITING_ON_BOX;
			ELSE
				// If vacuum was not achieved, then the side pick failed. Increment the fail counter
				SideFailureCount := SideFailureCount + 1;
				IF SideFailureCount = NUM_SIDE_TRIES THEN
					// If the side fails too many times, raise an error
					SideGrabFailAlarm := TRUE;
					state := SERVORAM_ERROR;
				ELSE
					// Otherwise, try again
					gIO.DOs.SidePickCylinder := TRUE;
					state := SERVORAM_PICK_SIDES;
				END_IF
			END_IF

		SERVORAM_WAITING_ON_BOX:
			// Run the delay timer when a box is seen
			RamDelayTimer.IN := gIO.DIs.BodyDetect;
			// When the delay finishes, move the ram to the end position
			IF gIO.DIs.SidePickVacuumAchieved AND RamDelayTimer.Q THEN
				gServoRamInterface.Parameters.MovementParameters.Position := gHMI.Parameters.ServoRamEndPosition;
				gServoRamInterface.Parameters.MovementParameters.Velocity := gHMI.Parameters.ServoRamBoxFormingVelocity;
				gRamAtStopPosition := FALSE;
				gServoRamInterface.Commands.RequestMoveAbs := TRUE;
				ServoRamBusy := TRUE ;
				gRamWaitingOnBox := FALSE;
				state := SERVORAM_TRIGGER_FOLD;
			ELSE
				IF NOT gIO.DIs.SidePickVacuumAchieved THEN
				SideGrabFailAlarm := TRUE;
				state := SERVORAM_ERROR;
			END_IF
		END_IF

		SERVORAM_TRIGGER_FOLD:
			IF gServoRamInterface.Status.ActualPosition > gHMI.Parameters.ServoRamFoldStartPos THEN
				gIO.DOs.FoldingHoldVacuum := TRUE;
				gIO.DOs.LeftSideFoldCylinder := TRUE;
				gIO.DOs.RightSideFoldCylinder := TRUE;
				state := SERVORAM_RELEASE_FOLD;
			END_IF

		SERVORAM_RELEASE_FOLD:
			IF gServoRamInterface.Status.ActualPosition > gHMI.Parameters.ServoRamFoldEndPos THEN
				gIO.DOs.LeftSideFoldCylinder := FALSE;
				gIO.DOs.RightSideFoldCylinder := FALSE;
				state := SERVORAM_MOVE_TO_END;
			END_IF

		SERVORAM_MOVE_TO_END:
			// When the move is complete, check if there is a configured dwell time
			IF gIO.DIs.SidePickVacuumAchieved AND gServoRamInterface.Status.MoveComplete THEN
				gServoRamInterface.Status.MoveComplete := FALSE;
				gRamAtStopPosition := TRUE;
				ServoRamBusy := FALSE;
				gServoRamInterface.Commands.ToMapp.Update := TRUE; //This forces update of the torque limit. This will be cleared automatically
				IF gHMI.Parameters.ServoRamEndDwellTime > 0 THEN
					// If there is a dwell time, execute the dwell
					EndDwellTimer.IN := TRUE;
					state := SERVORAM_DWELL_AT_END;
				ELSE
					// Otherwise, release the vaccuum and move back to the starting position
					gCyclesToFinish := gCyclesToFinish - 1;

					CycleCount := CycleCount + 1;
					LubeCount := LubeCount + 1;
					gIO.DOs.SidePanelVacOn := FALSE;
					gIO.DOs.SidePanelHoldVacuum := FALSE;
					gIO.DOs.FoldingHoldVacuum := FALSE;
					gIO.DOs.LeftSideFoldCylinder := FALSE;
					gIO.DOs.RightSideFoldCylinder := FALSE;
					gServoRamInterface.Parameters.MovementParameters.Position := gHMI.Parameters.ServoRamStartPosition;
					gServoRamInterface.Parameters.MovementParameters.Velocity := gHMI.Parameters.ServoRamNegativeVelocity;
					gServoRamInterface.Commands.RequestMoveAbs := TRUE;
					gRamAtStopPosition := FALSE;
					ServoRamBusy := TRUE;
					gRamWaitingOnBox := TRUE;
					state := SERVORAM_MOVE_TO_START;
				END_IF
				ELSE
					IF NOT gIO.DIs.SidePickVacuumAchieved THEN
					SideGrabFailAlarm := TRUE;
					state := SERVORAM_ERROR;
				END_IF
			END_IF

		SERVORAM_DWELL_AT_END:

			// Wait for the timer to finish
			EndDwellTimer.IN := TRUE;
			IF EndDwellTimer.Q THEN
				gCyclesToFinish := gCyclesToFinish - 1;

				// Release the vacuum and move back to the starting position
				EndDwellTimer.IN := FALSE;
				CycleCount := CycleCount + 1;
				LubeCount := LubeCount + 1;
				gIO.DOs.SidePanelVacOn := FALSE;
				gIO.DOs.SidePanelHoldVacuum := FALSE;
				gIO.DOs.FoldingHoldVacuum := FALSE;
				gIO.DOs.LeftSideFoldCylinder := FALSE;
				gIO.DOs.RightSideFoldCylinder := FALSE;
				gServoRamInterface.Parameters.MovementParameters.Position := gHMI.Parameters.ServoRamStartPosition;
				gServoRamInterface.Parameters.MovementParameters.Velocity := gHMI.Parameters.ServoRamNegativeVelocity;
				gServoRamInterface.Commands.RequestMoveAbs := TRUE;
				gRamAtStopPosition := FALSE;
				ServoRamBusy := TRUE;
				gRamWaitingOnBox := TRUE;
				state := SERVORAM_MOVE_TO_START;
			END_IF

			//these EX states are a copy the states above, but with no actuators being used and no evluation of inputs to know if it is OK to continue
		SERVORAM_MOVE_TO_START_EX:

			IF gServoRamInterface.Status.MoveComplete THEN
				gServoRamInterface.Status.MoveComplete := FALSE;
				ServoRamBusy := FALSE;
				IF NOT ExerciseRam THEN
					state := SERVORAM_IDLE;
				ELSE
					state := SERVORAM_PICK_SIDES_EX;
				END_IF

			END_IF

		SERVORAM_PICK_SIDES_EX:
			SidePickTimer.IN := TRUE;
			// Wait for the side pick timer, then retract the side pick
			IF SidePickTimer.Q THEN
				SidePickRetractTimer.IN := TRUE;
			END_IF
			// When the side pick is retracted, check for side panels
			IF SidePickRetractTimer.Q THEN
				SidePickTimer.IN := FALSE;
				SidePickRetractTimer.IN := FALSE;
				state := SERVORAM_CHECK_FOR_SIDES_EX;
			END_IF

		SERVORAM_CHECK_FOR_SIDES_EX:
			// If the side pick has vacuum, then the sides were picked, move to middle position
			gServoRamInterface.Parameters.MovementParameters.Position := gHMI.Parameters.ServoRamMiddlePosition;
			gServoRamInterface.Parameters.MovementParameters.Velocity := gHMI.Parameters.ServoRamSideFormingVelocity;
			gServoRamInterface.Commands.RequestMoveAbs := TRUE;
			state := SERVORAM_MOVE_TO_MIDDLE_EX;

		SERVORAM_MOVE_TO_MIDDLE_EX:
			// When the ram gets to the middle position, extend the folders
			IF gServoRamInterface.Status.MoveComplete THEN
				gServoRamInterface.Status.MoveComplete := FALSE;
				state := SERVORAM_FOLD_SIDES_EX;
			END_IF

		SERVORAM_FOLD_SIDES_EX:
			SideFoldTimer.IN := TRUE;
			// Wait for the side fold timer, then retract the side folders
			IF SideFoldTimer.Q THEN
				SideFoldRetractTimer.IN := TRUE;
			END_IF
			// When the side fold is retracted, check that the fold was successful
			IF SideFoldRetractTimer.Q THEN
				state := SERVORAM_CHECK_FOR_FOLDS_EX;
			END_IF

		SERVORAM_CHECK_FOR_FOLDS_EX:
			state := SERVORAM_WAITING_ON_BOX_EX;

		SERVORAM_WAITING_ON_BOX_EX:
			RamDelayTimer.IN := TRUE;
			// When the delay finishes, move the ram to the end position
			IF RamDelayTimer.Q THEN
				gServoRamInterface.Parameters.MovementParameters.Position := gHMI.Parameters.ServoRamEndPosition;
				gServoRamInterface.Parameters.MovementParameters.Velocity := gHMI.Parameters.ServoRamBoxFormingVelocity;
				gServoRamInterface.Commands.RequestMoveAbs := TRUE;
				state := SERVORAM_MOVE_TO_END_EX;
			END_IF

		SERVORAM_MOVE_TO_END_EX:
			// When the move is complete, check if there is a configured dwell time
			IF gServoRamInterface.Status.MoveComplete THEN
				gServoRamInterface.Status.MoveComplete := FALSE;
				IF gHMI.Parameters.ServoRamEndDwellTime > 0 THEN
					// If there is a dwell time, execute the dwell
					EndDwellTimer.IN := TRUE;
					state := SERVORAM_DWELL_AT_END_EX;
				ELSE
					// Otherwise, release the vaccuum and move back to the starting position
					CycleCount := CycleCount + 1;
					LubeCount := LubeCount + 1;
					gServoRamInterface.Parameters.MovementParameters.Position := gHMI.Parameters.ServoRamStartPosition;
					gServoRamInterface.Parameters.MovementParameters.Velocity := gHMI.Parameters.ServoRamNegativeVelocity;
					gServoRamInterface.Commands.RequestMoveAbs := TRUE;
					state := SERVORAM_MOVE_TO_START_EX;
				END_IF
			END_IF

		SERVORAM_DWELL_AT_END_EX:

			// Wait for the timer to finish
			EndDwellTimer.IN := TRUE;
			IF EndDwellTimer.Q THEN
				// Release the vacuum and move back to the starting position
				EndDwellTimer.IN := FALSE;
				CycleCount := CycleCount + 1;
				LubeCount := LubeCount + 1;
				gServoRamInterface.Parameters.MovementParameters.Position := gHMI.Parameters.ServoRamStartPosition;
				gServoRamInterface.Parameters.MovementParameters.Velocity := gHMI.Parameters.ServoRamNegativeVelocity;
				gServoRamInterface.Commands.RequestMoveAbs := TRUE;
				state := SERVORAM_MOVE_TO_START_EX;
			END_IF

		SERVORAM_ERROR:

			gCyclesToFinish := 0;

			ServoRamAutoHome := FALSE;
			gServoRamInterface.Status.MoveComplete := FALSE;
			gHMI.Commands.CycleServoRam := FALSE;
			ServoRamBusy := FALSE;
			ServoRamAutoHome := FALSE;
			gIO.DOs.SidePanelHoldVacuum := FALSE;
			gIO.DOs.LeftSideFoldCylinder := FALSE;
			gIO.DOs.RightSideFoldCylinder := FALSE;
			gIO.DOs.SidePickCylinder := FALSE;
			gIO.DOs.SidePanelHoldVacuum := FALSE;
			gIO.DOs.BodyVacuumOn := FALSE;
			gIO.DOs.FoldingHoldVacuum := FALSE;
			gRamWaitingOnBox := FALSE;

			IF (gNumActiveAlarms = 0) THEN
				SideFailureCount := 0;
				FoldFailureCount := 0;
				state := SERVORAM_WAIT_FOR_HOME;
			END_IF

	END_CASE;

	// FUB Calls
	EndDwellTimer.PT := gHMI.Parameters.ServoRamEndDwellTime; //Use existing dwell time from HMI
	EndDwellTimer();
	SidePickTimer.PT := gHMI.Parameters.ServoRamSidePickTime;
	SidePickTimer();
	SidePickRetractTimer.PT := gHMI.Parameters.ServoRamSidePickRetractTime;
	SidePickRetractTimer();
	SideFoldTimer.PT := gHMI.Parameters.ServoRamSideFoldTime;
	SideFoldTimer();
	SideFoldRetractTimer.PT := gHMI.Parameters.ServoRamSideFoldRetractTime;
	SideFoldRetractTimer();
	RamDelayTimer.PT := gHMI.Parameters.RamDelay;
	RamDelayTimer();
	ResetTimeoutTimer.PT := gHMI.Parameters.ServoRamTimeoutTime;
	ResetTimeoutTimer();

END_PROGRAM

PROGRAM _EXIT
				(* Insert code here *)

END_PROGRAM
```

### Program Logical/ServoMotion/ServoPnPHandler (IEC)

#### Main.st
```iecst
PROGRAM _INIT

	// Velocities and Accels
	gHMI.Parameters.ServoPnPJogVelocity := 10;
	gHMI.Parameters.ServoPnPPositiveVelocity := 90.0;
	gHMI.Parameters.ServoPnPNegativeVelocity := 90.0;
	gHMI.Parameters.ServoPnPAccel := 1000.0;

	// Positions
	gHMI.Parameters.ServoPnPStartPosition := 0;
	gHMI.Parameters.ServoPnPVacuumOffPosition := 80; //this is the position where the vacuum will be turned off on the way down to horizontal
	gHMI.Parameters.ServoPnPEndPosition := 100; //105 was the original position. Found that the box was rubbing the suction cups

	// Times
	gHMI.Parameters.ServoPnPStartDwellTime := 100;
	gHMI.Parameters.BodyKickerTime := 250;			//500 is original setting
	gHMI.Parameters.BodyKickerRetractTime := 100;	//500 is original setting

	// Other
	gHMI.Parameters.ServoPnPTorqueLimit := 8.0;	//3 is original setting.
	//Made adjustments for running 20-22 BPM 01-17-2025
END_PROGRAM

PROGRAM _CYCLIC

	IF gHighSeverityAlarmActive THEN
		state := SERVOPNP_ERROR;
	END_IF

	StartDwellTimer.IN := FALSE; //Set in state machine if needed
	BodyKickerTimer.IN := FALSE;
	BodyKickerRetractTimer.IN := FALSE;

//	IF (NOT gHMI.Commands.CycleServoPnP AND NOT SingleCyclePnP) AND state <> SERVOPNP_ERROR AND gServoPnPInterface.Status.Homed THEN
//		state := SERVOPNP_IDLE;
//	END_IF

	// Resetting clears the grab alarm
	IF gHMI.Commands.RequestReset THEN
		BodyGrabFailAlarm := FALSE;
	END_IF

	CASE state OF

		SERVOPNP_WAIT_FOR_HOME:

            // Pick and place should home automatically on machine start up.
			IF gServoPnPInterface.Status.Homed AND ServoPnPFirstHomeExecuted THEN
				ServoPnPAutoHome := FALSE;
				gPnPAtStopPosition := TRUE;
				gHMI.Commands.CycleServoPnP := FALSE;
				gServoPnPInterface.Commands.ToMapp.TorqueLimitingOn := TRUE; //turn torque limiting on
				state := SERVOPNP_IDLE;
			ELSIF gServoPnPInterface.Status.PoweredOn AND NOT ServoPnPFirstHomeExecuted THEN
                ServoPnPAutoHome := TRUE;
                //GuideCylinder    := FALSE;
				state := SERVOPNP_WAIT_FOR_AUTO_HOME;
			END_IF

		SERVOPNP_WAIT_FOR_AUTO_HOME:

			IF gServoPnPInterface.Status.Homed AND ServoPnPFirstHomeExecuted THEN
				ServoPnPAutoHome := FALSE;
				gPnPAtStopPosition := TRUE;
				gHMI.Commands.CycleServoPnP := FALSE;
				gServoPnPInterface.Commands.ToMapp.TorqueLimitingOn := TRUE; //turn torque limiting on
				state := SERVOPNP_IDLE;
			END_IF

		SERVOPNP_IDLE:

			ServoPnPAutoHome := FALSE;
			gServoPnPInterface.Status.MoveComplete := FALSE;

            // Wait for the run command, then go to the start position
			IF (gHMI.Commands.CycleServoPnP OR (SingleCyclePnP)) AND ServoPnPFirstHomeExecuted THEN
				gCyclesToFinish := gCyclesToFinish + 1;
				gServoPnPInterface.Parameters.MovementParameters.Position := gHMI.Parameters.ServoPnPStartPosition;
				gServoPnPInterface.Parameters.MovementParameters.Velocity := gHMI.Parameters.ServoPnPPositiveVelocity;
				gServoPnPInterface.Commands.RequestMoveAbs := TRUE;
				state := SERVOPNP_MOVE_TO_HOPPER;
			END_IF

		SERVOPNP_MOVE_TO_HOPPER:

            GuideCylinder    := FALSE;

			// At the hopper position, if the body hopper is on, turn on the vacuum and dwell if there is a dwell time, or move to horizontal
			IF gServoPnPInterface.Status.MoveComplete AND gIO.DIs.BodyHopperMotor_RUN THEN
				gIO.DOs.BodyVacuumOn := TRUE;
				gServoPnPInterface.Status.MoveComplete := FALSE;
				IF gHMI.Parameters.ServoPnPStartDwellTime > 0 THEN
					state := SERVOPNP_DWELL_AT_HOPPER;
				ELSE
					gServoPnPInterface.Parameters.MovementParameters.Position := gHMI.Parameters.ServoPnPEndPosition;
					gServoPnPInterface.Parameters.MovementParameters.Velocity := gHMI.Parameters.ServoPnPNegativeVelocity;
					gServoPnPInterface.Commands.RequestMoveAbs := TRUE;
					state := SERVOPNP_MOVE_TO_HORIZONTAL;
				END_IF
			END_IF

		SERVOPNP_DWELL_AT_HOPPER:

            // Wait for the timer to finish, then start the move towards horizontal
            StartDwellTimer.IN := TRUE;
			IF StartDwellTimer.Q THEN
				StartDwellTimer.IN := FALSE;
				gServoPnPInterface.Parameters.MovementParameters.Position := gHMI.Parameters.ServoPnPEndPosition;
				gServoPnPInterface.Parameters.MovementParameters.Velocity := gHMI.Parameters.ServoPnPNegativeVelocity;
				gServoPnPInterface.Commands.RequestMoveAbs := TRUE;
				state := SERVOPNP_CHECK_FOR_BOX;
			END_IF

		SERVOPNP_CHECK_FOR_BOX:

			// After rotating 20 degrees, check that a box is actually grabbed
			IF gServoPnPInterface.Status.ActualPosition > 20 THEN
				IF gIO.DIs.BodyVacuumAchieved THEN
					// If the vacuum was achieved, then continue the move to horizontal
					FailureCount := 0;
					state := SERVOPNP_MOVE_TO_HORIZONTAL;
				ELSE
					FailureCount := FailureCount + 1;
					// If the vacuum failed, a box was not grabbed. Unless this was the third failure, try again
					IF FailureCount = NUM_PNP_TRIES THEN
						BodyGrabFailAlarm := TRUE;
						// Return home
						gServoPnPInterface.Parameters.MovementParameters.Position := gHMI.Parameters.ServoPnPStartPosition;
						gServoPnPInterface.Parameters.MovementParameters.Velocity := gHMI.Parameters.ServoPnPPositiveVelocity;
						gServoPnPInterface.Commands.RequestMoveAbs := TRUE;
						state := SERVOPNP_ERROR;
                    ELSE
						state := SERVOPNP_ABORT_AND_RETURN;
					END_IF
				END_IF
			END_IF

		SERVOPNP_MOVE_TO_HORIZONTAL:

			IF gServoPnPInterface.Status.ActualPosition > gHMI.Parameters.ServoPnPVacuumOffPosition THEN
				gIO.DOs.BodyVacuumOn := FALSE;
			END_IF

			// At the horizontal position, cut off the vacuum
			IF gServoPnPInterface.Status.MoveComplete THEN
				gIO.DOs.BodyVacuumOn := FALSE;
				// Wait for the ram to be ready (sucessful side folds) then push the box to the feeder and wait for it to clear
				IF (SingleCyclePnP) THEN
					SingleCyclePnP := FALSE;
					state := SERVOPNP_IDLE;
				ELSIF (*gIO.DIs.SideFoldVacuumAchieved AND *) gServoRamInterface.Status.ClearOfRoller AND gRamWaitingOnBox THEN
					gServoPnPInterface.Status.MoveComplete := FALSE;
					gIO.DOs.BodyKicker := TRUE;
					state := SERVOPNP_REMOVE_BOX;
				END_IF
			END_IF

        SERVOPNP_REMOVE_BOX:

            GuideCylinder := TRUE;
			// After the delay, turn off the kicker and start the retract timer
			BodyKickerTimer.IN := TRUE;
			IF BodyKickerTimer.Q THEN
				gIO.DOs.BodyKicker := FALSE;
				BodyKickerRetractTimer.IN := TRUE;
			END_IF
			// When the retract timer is done and the adhesive photoeye falls, send the pick and place home
			FTrig_AdhesivePhotoeye(CLK:=gIO.DIs.AdhesivePhotoEye);
			IF FTrig_AdhesivePhotoeye.Q AND BodyKickerRetractTimer.Q THEN
				BodyKickerTimer.IN := FALSE;
				BodyKickerRetractTimer.IN := FALSE;

				IF (NOT gHMI.Commands.CycleServoPnP) THEN
					state := SERVOPNP_IDLE;
				ELSE
					// On the falling edge of the adhesive photoeye, send the pick and place back to the hopper
					gCyclesToFinish := gCyclesToFinish + 1;
					gServoPnPInterface.Parameters.MovementParameters.Position := gHMI.Parameters.ServoPnPStartPosition;
					gServoPnPInterface.Parameters.MovementParameters.Velocity := gHMI.Parameters.ServoPnPPositiveVelocity;
                    gServoPnPInterface.Commands.RequestMoveAbs := TRUE;
                    //GuideCylinder := TRUE;
					state := SERVOPNP_MOVE_TO_HOPPER;
				END_IF
			END_IF

        SERVOPNP_ABORT_AND_RETURN:
            IF gServoPnPInterface.Status.MoveComplete THEN
                gServoPnPInterface.Status.MoveComplete := FALSE;
                gServoPnPInterface.Parameters.MovementParameters.Position := gHMI.Parameters.ServoPnPStartPosition;
                gServoPnPInterface.Parameters.MovementParameters.Velocity := gHMI.Parameters.ServoPnPNegativeVelocity;
                gServoPnPInterface.Commands.RequestMoveAbs := TRUE;
                state := SERVOPNP_MOVE_TO_HOPPER;
            END_IF

		SERVOPNP_ERROR:
            // Error response
			gServoPnPInterface.Status.MoveComplete := FALSE;
			gHMI.Commands.CycleServoPnP := FALSE;
			ServoPnPAutoHome := FALSE;
			gServoPnPInterface.Commands.RequestMoveAbs := FALSE;
			gIO.DOs.BodyVacuumOn := FALSE;
			gIO.DOs.BodyKicker := FALSE;
			SingleCyclePnP := FALSE;
			IF (gNumActiveAlarms = 0) THEN
				FailureCount := 0;
				state := SERVOPNP_WAIT_FOR_HOME;
			END_IF

	END_CASE;

	//The kicker is not allowed to be on if the servo PNP is below 97 degrees (Smaller number => further from horizontal)
	IF gServoPnPInterface.Status.ActualPosition < 97.0 THEN
		gIO.DOs.BodyKicker := FALSE;
	END_IF

	StartDwellTimer.PT := gHMI.Parameters.ServoPnPStartDwellTime;
	StartDwellTimer();
	BodyKickerTimer.PT := gHMI.Parameters.BodyKickerTime;
	BodyKickerTimer();
	BodyKickerRetractTimer.PT := gHMI.Parameters.BodyKickerRetractTime;
    BodyKickerRetractTimer();

//    IF gForceBodyKicker THEN
//        gIO.DOs.BodyKicker := TRUE;
//    ELSE
//        gIO.DOs.BodyKicker := FALSE;
//    END_IF

	END_PROGRAM

PROGRAM _EXIT
				(* Insert code here *)

				END_PROGRAM
```

### Program Logical/ServoMotion/ServoFeedHandler (IEC)

#### Main.st
```iecst
PROGRAM _INIT
	(* Insert code here *)

    gHMI.Parameters.ServoFeedJogVelocity := 50;
    gHMI.Parameters.ServoFeedVelocity := 600.0;
    gHMI.Parameters.ServoFeedAccel := 600.0;
    HoperLowStop;

END_PROGRAM

PROGRAM _CYCLIC

//	IF gNumActiveAlarms  > 0 THEN
//		state := SERVOFEED_ERROR;
//	END_IF

    IF gHighSeverityAlarmActive THEN
        state := SERVOFEED_ERROR;
    END_IF

    CASE state OF

        SERVOFEED_WAIT_FOR_HOME:

            //servo ram should home automatically on machine start up. This is a direct home axis and should not rquire a home command
            IF gServoFeedInterface.Status.Homed THEN
                state := SERVOFEED_IDLE;
            END_IF

        SERVOFEED_IDLE:

            IF gHMI.Commands.StartServoFeed AND ServoFeedFirstHomeExecuted THEN

                gServoFeedInterface.Commands.RequestMoveVelocity := TRUE;

                state := SERVOFEED_MOVE_VELOCITY;
            END_IF

        SERVOFEED_MOVE_VELOCITY:

            //Added gDownstreamBlocked := TRUE. 07-14-22.
            IF (gHMI.Commands.StartServoFeed = FALSE AND gCyclesToFinish = 0) OR gDownstreamBlocked = TRUE THEN
                gServoFeedInterface.Commands.RequestMoveVelocity := FALSE;

                state := SERVOFEED_IDLE;
                //                END_IF
            END_IF

        SERVOFEED_ERROR:

            gServoFeedInterface.Status.MoveComplete := FALSE;
            gHMI.Commands.StartServoFeed := FALSE;

            gServoFeedInterface.Commands.RequestMoveVelocity := FALSE;

            IF (gNumActiveAlarms = 0) THEN
                state := SERVOFEED_WAIT_FOR_HOME;
            END_IF

    END_CASE;
	FeedStopTimer();
END_PROGRAM

PROGRAM _EXIT
				(* Insert code here *)

END_PROGRAM
```

### Program Logical/ServoMotion/LeftHopperHandler (IEC)

#### Main.st
```iecst
PROGRAM _INIT
	(* Insert code here *)

	gHMI.Parameters.LeftHopperJogVelocity := 3.35;
	gHMI.Parameters.LeftHopperVelocity := 3.35;
	gHMI.Parameters.LeftHopperAccel := 180.0;

	gHMI.Parameters.LeftHopperTorqueLimit := 1.0;

	gHMI.Parameters.LeftHopperDwellTime := 1500; //1 s
	gHMI.Parameters.AtTorqueTime := 500; //1 s

	gHMI.Parameters.LeftHopperTimeoutTime := 600000; //10 minutes

END_PROGRAM

PROGRAM _CYCLIC

	IF gNumActiveAlarms  > 0 THEN
		state := SERVOHOPPER_ERROR;
	END_IF

	IF gHighSeverityAlarmActive THEN
		state := SERVOHOPPER_ERROR;
	END_IF

	//make sure that torque limiting is turned on while jogging
	//	IF EDGEPOS(gHMI.Commands.JogLeftHopperPos) THEN
	//		gLeftHopperInterface.Commands.ToMapp.TorqueLimitingOn := TRUE;
	//	END_IF
	//	IF EDGEPOS(gHMI.Commands.JogLeftHopperNeg) THEN
	//		gLeftHopperInterface.Commands.ToMapp.TorqueLimitingOn := TRUE;
	//	END_IF

	StartDwellTimer.IN := FALSE; //clear otuside state machine. will be set true in appropriate state
	AtTorqueTimer.IN := FALSE;
	ResetTimeoutTimer.IN := FALSE;

	// If the hopper has been reset but the machine isn't running, only let the hopper run for an alotted time to protect the motor
	IF gIO.DIs.LeftHopperMotor_RUN AND NOT gLeftHopperInterface.Status.Error AND (NOT gHMI.Commands.RequestVFDRun) THEN
		ResetTimeoutTimer.IN := TRUE;
	END_IF
	IF ResetTimeoutTimer.Q THEN
		ResetTimeoutAlarm := TRUE;
	END_IF

	// Resetting clears the timeout alarms
	IF gHMI.Commands.RequestReset THEN
		ResetTimeoutAlarm := FALSE;
	END_IF

	CASE state OF

		SERVOHOPPER_WAIT_FOR_HOME:

			//servo ram should home automatically on machine start up. This is a direct home axis and should not rquire a home command
			IF gServoFeedInterface.Status.Homed THEN
				gLeftHopperInterface.Commands.ToMapp.TorqueLimitingOn := TRUE;
				state := SERVOHOPPER_IDLE;
			END_IF

		SERVOHOPPER_IDLE:

			IF gIO.DIs.LeftHopperMotor_RUN AND LeftHopperFirstHomeExecuted THEN
				gLeftHopperInterface.Commands.ToMapp.TorqueLimitingOn := TRUE; //turn torque limiting on

				gLeftHopperInterface.Commands.RequestMoveVelocity := TRUE;
				gLeftHopperInterface.Parameters.MovementParameters.Direction := 0;

				state := SERVOHOPPER_MOVE_VELOCITY;
			END_IF

		SERVOHOPPER_MOVE_VELOCITY:

			AtTorqueTimer.IN := (gLeftHopperInterface.Status.ActualTorque >= gHMI.Parameters.LeftHopperTorqueLimit *0.90);

			IF gIO.DIs.LeftHopperMotor_OFF = TRUE THEN
				gLeftHopperInterface.Commands.RequestMoveVelocity := FALSE;
				state := SERVOHOPPER_IDLE;
			ELSIF AtTorqueTimer.Q THEN
				gLeftHopperInterface.Parameters.MovementParameters.Direction := 1;
				gLeftHopperInterface.Commands.ToMapp.Update := TRUE;
				gLeftHopperInterface.Commands.RequestMoveVelocity := TRUE;
				state := SERVOHOPPER_COOLDOWN;
			END_IF

		SERVOHOPPER_COOLDOWN:

			StartDwellTimer.IN := TRUE;

			IF gIO.DIs.LeftHopperMotor_OFF = TRUE THEN
				gLeftHopperInterface.Commands.RequestMoveVelocity := FALSE;
				state := SERVOHOPPER_IDLE;
			ELSIF StartDwellTimer.Q THEN
//				gLeftHopperInterface.Parameters.MovementParameters.Direction := 0;
				gLeftHopperInterface.Commands.ToMapp.Update := TRUE;
				gLeftHopperInterface.Commands.RequestMoveVelocity := TRUE;
				state := SERVOHOPPER_MOVE_VELOCITY;
			END_IF

		SERVOHOPPER_ERROR:

			gLeftHopperInterface.Status.MoveComplete := TRUE;
			gHMI.Commands.StartLeftHopper := FALSE;

			gLeftHopperInterface.Commands.RequestMoveVelocity := FALSE;

			ResetTimeoutTimer.IN := FALSE;

			IF (gNumActiveAlarms = 0) THEN
				state := SERVOHOPPER_WAIT_FOR_HOME;
			END_IF

	END_CASE;

	StartDwellTimer.PT := gHMI.Parameters.LeftHopperDwellTime; //500 ms
	StartDwellTimer();
	AtTorqueTimer.PT := gHMI.Parameters.AtTorqueTime; //500 ms
	AtTorqueTimer();
	ResetTimeoutTimer.PT := gHMI.Parameters.LeftHopperTimeoutTime;
	ResetTimeoutTimer();

END_PROGRAM

PROGRAM _EXIT
				(* Insert code here *)

END_PROGRAM
```

### Program Logical/ServoMotion/RightHopperHandler (IEC)

#### Main.st
```iecst
PROGRAM _INIT
	(* Insert code here *)

	gHMI.Parameters.RightHopperJogVelocity := 3.35;
	gHMI.Parameters.RightHopperVelocity := 3.35;
	gHMI.Parameters.RightHopperAccel := 180.0;

	gHMI.Parameters.RightHopperTorqueLimit := 1.0;

	gHMI.Parameters.RightHopperDwellTime := 1500; //1 s
	gHMI.Parameters.AtTorqueTime := 500; //1 s

	gHMI.Parameters.RightHopperTimeoutTime := 600000;

END_PROGRAM

PROGRAM _CYCLIC

	IF gNumActiveAlarms  > 0 THEN
		state := SERVOHOPPER_ERROR;
	END_IF

	IF gHighSeverityAlarmActive THEN
		state := SERVOHOPPER_ERROR;
	END_IF

	//make sure that torque limiting is turned on while jogging
	//	IF EDGEPOS(gHMI.Commands.JogRightHopperPos) THEN
	//		gRightHopperInterface.Commands.ToMapp.TorqueLimitingOn := TRUE;
	//	END_IF
	//	IF EDGEPOS(gHMI.Commands.JogRightHopperNeg) THEN
	//		gRightHopperInterface.Commands.ToMapp.TorqueLimitingOn := TRUE;
	//	END_IF

	StartDwellTimer.IN := FALSE; //clear otuside state machine. will  e set true in appropriate state
	AtTorqueTimer.IN := FALSE;
	ResetTimeoutTimer.IN := FALSE;

	// If the hopper has been reset but the machine isn't running, only let the hopper run for an alotted time to protect the motor
	IF gIO.DIs.RightHopperMotor_RUN AND NOT gLeftHopperInterface.Status.Error AND (NOT gHMI.Commands.RequestVFDRun) THEN
		ResetTimeoutTimer.IN := TRUE;
	END_IF
	IF ResetTimeoutTimer.Q THEN
		ResetTimeoutAlarm := TRUE;
	END_IF

	// Resetting clears the timeout alarms
	IF gHMI.Commands.RequestReset THEN
		ResetTimeoutAlarm := FALSE;
	END_IF

	CASE state OF

		SERVOHOPPER_WAIT_FOR_HOME:

			//servo ram should home automatically on machine start up. This is a direct home axis and should not rquire a home command
			IF gServoFeedInterface.Status.Homed THEN
				gRightHopperInterface.Commands.ToMapp.TorqueLimitingOn := TRUE;
				state := SERVOHOPPER_IDLE;
			END_IF

		SERVOHOPPER_IDLE:

			IF gIO.DIs.RightHopperMotor_RUN AND RightHopperFirstHomeExecuted THEN
				gRightHopperInterface.Commands.ToMapp.TorqueLimitingOn := TRUE; //turn torque limiting on

				gRightHopperInterface.Commands.RequestMoveVelocity := TRUE;
				gRightHopperInterface.Parameters.MovementParameters.Direction := 0;

				state := SERVOHOPPER_MOVE_VELOCITY;
			END_IF

		SERVOHOPPER_MOVE_VELOCITY:

			AtTorqueTimer.IN := (gRightHopperInterface.Status.ActualTorque >= gHMI.Parameters.RightHopperTorqueLimit *0.90);

			IF gIO.DIs.RightHopperMotor_OFF = TRUE THEN
				gRightHopperInterface.Commands.RequestMoveVelocity := FALSE;
				state := SERVOHOPPER_IDLE;
			ELSIF AtTorqueTimer.Q THEN
//				gRightHopperInterface.Parameters.MovementParameters.Direction := 1;
				gRightHopperInterface.Commands.ToMapp.Update := TRUE;
				gRightHopperInterface.Commands.RequestMoveVelocity := TRUE;
				state := SERVOHOPPER_COOLDOWN;
			END_IF

		SERVOHOPPER_COOLDOWN:

			StartDwellTimer.IN := TRUE;

			IF gIO.DIs.RightHopperMotor_OFF = TRUE THEN
				gRightHopperInterface.Commands.RequestMoveVelocity := FALSE;
				state := SERVOHOPPER_IDLE;
			ELSIF StartDwellTimer.Q THEN
				gRightHopperInterface.Parameters.MovementParameters.Direction := 0;
				gRightHopperInterface.Commands.ToMapp.Update := TRUE;
				gRightHopperInterface.Commands.RequestMoveVelocity := TRUE;
				state := SERVOHOPPER_MOVE_VELOCITY;
			END_IF

		SERVOHOPPER_ERROR:

			gRightHopperInterface.Status.MoveComplete := TRUE;
			gHMI.Commands.StartRightHopper := FALSE;

			gRightHopperInterface.Commands.RequestMoveVelocity := FALSE;

			ResetTimeoutTimer.IN := FALSE;

			IF (gNumActiveAlarms = 0) THEN
				state := SERVOHOPPER_WAIT_FOR_HOME;
			END_IF

	END_CASE;

	StartDwellTimer.PT := gHMI.Parameters.RightHopperDwellTime; //500 ms
	StartDwellTimer();
	AtTorqueTimer.PT := gHMI.Parameters.AtTorqueTime; //500 ms
	AtTorqueTimer();
	ResetTimeoutTimer.PT := gHMI.Parameters.RightHopperTimeoutTime;
	ResetTimeoutTimer();

END_PROGRAM

PROGRAM _EXIT
				(* Insert code here *)

END_PROGRAM
```

### Program Logical/ServoMotion/MappCalls (IEC)

#### Variables.var - Local variables
```iecst
VAR
	BodyHopper : AxisBasic;
	LeftHopper : AxisBasic;
	RightHopper : AxisBasic;
	ServoFeed : AxisBasic;
	ServoRam : AxisBasic;
	ServoPnP : AxisBasic;
	ServoOverride : REAL := 1.0;
END_VAR
```

### Program Logical/ServoMotion/MotionHandler (ANSIC)

#### Variables.var
```iecst
VAR
	ServoFeedHandler : AxisHandler;
	ServoPnPHandler : AxisHandler;
	BodyHopperHandler : AxisHandler;
	LeftHopperHandler : AxisHandler;
	RightHopperHandler : AxisHandler;
	ServoRamHandler : AxisHandler;
	OldTorqueLimitBodyHopper : REAL;
	OldTorqueLimitLeftHopper : REAL;
	OldTorqueLimitRightHopper : REAL;
	OldTorqueLimitFeed : REAL;
	OldTorqueLimitRam : REAL;
	SetHardwareInputs : MC_BR_SetHardwareInputs;
	PowerSaverTime : TIME;
	PowerSaverTimer : TON;
END_VAR
```
